// TIA Portal project "Clasificacion de Piezas" (V16)

(* hardware
DEVICE "S71500/ET200MP station_1"  S7-1500 station
   slot 0: "Perfil soporte_0"  Rack  6ES7 590-1***0-0AA0
   slot 1: "PLC_1"  CPU 1512C-1 PN  6ES7 512-1CK00-0AB0  V2.8
      slot 3: "Display de la CPU_1"  6ES7591-1AA00-0AA0
      slot 32768: "Interfaz PROFINET_1"  X1
         slot 32769: "Puerto_1"  X1 P1
         slot 32770: "Puerto_2"  X1 P2
      slot 34817: "Virtual CP interface port_1"  Virtual CP interface port  Virtual CP interface port
DEVICE "HMI_Clasificacion"  KTP900 Basic PN
   slot 0: "HMI_Clasificacion"  KTP900 Basic PN  6AV2 123-2JB03-0AX0  16.0.0.0
   slot 1: "HMI_RT_2"  KTP900 Basic PN  6AV2 123-2JB03-0AX0  16.0.0.0
   slot 5: "HMI_Clasificacion.IE_CP_1"  PROFINET Interface  16.0.0.0
      slot 1: "Interfaz PROFINET_1"  PROFINET Interface
         slot 1: "Port_1"  Port
*)

// ===== PLC "PLC_1"  CPU 1512C-1 PN =====

VAR_GLOBAL   // PLC tag table "Entradas"
   "PM" AT %M0.0 : Bool;   // Pulsador de Macha
   "PP" AT %M0.1 : Bool;   // Pulsador de Paro
   "SE" AT %M0.2 : Bool;   // Seta de Emergencia
   "PR" AT %M0.3 : Bool;   // Pulsador de Rearme
   "FCSuperior" AT %M0.4 : Bool;   // Final de Carrera Superior
   "FCInferior" AT %M0.5 : Bool;   // Final de Carrera Inferior
   "SenCintaEntrada" AT %M0.6 : Bool;   // Sensor de la Cinta de Entrada
   "SenCaja01PosIni" AT %M0.7 : Bool;   // Sensor de la Posición Inicial de la Caja 01
   "SenCaja02PosIni" AT %M1.0 : Bool;   // Sensor de la Posición Inicial de la Caja 02
   "SenCil01Rec" AT %M1.1 : Bool;   // Sensor del Cilindro Recogido
   "SenCil01Med" AT %M1.2 : Bool;   // Sensor del Cilindro en el Medio
   "SenCil01Ext" AT %M1.3 : Bool;   // Sensor del Cilindro Extendido
   "SenIndCaja01" AT %M1.4 : Bool;   // Sensor Inductivo de Giro de la Caja 01
   "SenIndCaja02" AT %M1.5 : Bool;   // Sensor Inductivo de Giro de la Caja 02
   "SenCinta01" AT %M1.6 : Bool;   // Sensor de la Cinta 01
   "SenCinta02" AT %M1.7 : Bool;   // Sensor de la Cinta 02
   "PMAux" AT %M2.0 : Bool;
   "PPAux" AT %M2.1 : Bool;
   "PRAux" AT %M2.2 : Bool;
   "Marcha" AT %M4.4 : Bool;
   "Paro" AT %M4.5 : Bool;
   "Rearme" AT %M4.6 : Bool;
END_VAR

VAR_GLOBAL   // PLC tag table "Salidas"
   "MotorVolteoCaja01Izq" AT %Q0.0 : Bool;   // Motor de Volteo hacia la Izquierda de La Caja 01
   "MotorVolteoCaja01Dch" AT %Q0.1 : Bool;   // Motor de Volteo hacia la Derecha de La Caja 01
   "MotorVolteoCaja02Izq" AT %Q0.2 : Bool;   // Motor de Volteo hacia la Izquierda de La Caja 02
   "MotorVolteoCaja02Dch" AT %Q0.3 : Bool;   // Motor de Volteo hacia la Derecha de La Caja 02
   "MotorCilindroRec" AT %Q0.4 : Bool;   // Motor de Recogida del Cilindro
   "MotorCilindroExt" AT %Q0.5 : Bool;   // Motor de Extension del Cilindro
   "MotorCinta01" AT %Q0.6 : Bool;   // Motor de la Cinta 01
   "MotorCinta02" AT %Q0.7 : Bool;   // Motor de la Cinta 02
   "MotorCintaEntradaAdelante" AT %Q1.0 : Bool;   // Motor de Avance de la Cinta de Entrada
   "MotorCintaEntradaAtras" AT %Q1.1 : Bool;   // Motor de Retroceso de la Cinta de Entrada
   "LV" AT %Q1.2 : Bool;   // Luz Verde
   "LN" AT %Q1.3 : Bool;   // Luz Naranja
   "LR" AT %Q1.4 : Bool;   // Luz Roja
   "LE" AT %Q1.5 : Bool;   // Luz de Emergencia
   "Sirena" AT %Q1.6 : Bool;   // Sirena
END_VAR

VAR_GLOBAL   // PLC tag table "Memorias"
   "Inicio" AT %M2.4 : Bool;
   "SolCondIni" AT %M2.5 : Bool;
   "IniCondIni" AT %M2.6 : Bool;
   "FinCondIni" AT %M2.7 : Bool;
   "ProdNorm" AT %M3.0 : Bool;
   "ParoFC" AT %M3.1 : Bool;
   "InicioCintaEntrada" AT %M3.2 : Bool;
   "InicioRecPiezas" AT %M3.3 : Bool;
   "InicioCinta1" AT %M3.4 : Bool;
   "InicioCinta2" AT %M3.5 : Bool;
   "SolMarchaFin" AT %M3.6 : Bool;
   "IniMarchaFin" AT %M3.7 : Bool;
   "FinMarchaFin" AT %M4.0 : Bool;
   "Emergencia" AT %M4.1 : Bool;
   "PararCintaEntrada" AT %M4.3 : Bool;
   "Timer1" AT %M4.7 : Bool;
   "Cont01" AT %M5.0 : Bool;
   "Cont02" AT %M5.1 : Bool;
   "Timer2" AT %M5.2 : Bool;
   "Timer3" AT %M5.3 : Bool;
   "Timer4" AT %M5.4 : Bool;
END_VAR

DATA_BLOCK "Sec_Principal_DB"   // DB1
{ S7_Optimized_Access := 'TRUE' }
VERSION : 0.1
// stored: InstanceOfName Sec_Principal
"Sec_Principal"
BEGIN
END_DATA_BLOCK

DATA_BLOCK "Recoger_Piezas_DB"   // DB2
{ S7_Optimized_Access := 'TRUE' }
VERSION : 0.1
// stored: InstanceOfName Recoger_Piezas
"Recoger_Piezas"
BEGIN
END_DATA_BLOCK

DATA_BLOCK "Marcha_Fin_DB"   // DB3
{ S7_Optimized_Access := 'TRUE' }
VERSION : 0.1
// stored: InstanceOfName Marcha_Fin
"Marcha_Fin"
BEGIN
END_DATA_BLOCK

DATA_BLOCK "Cond_Ini_DB"   // DB4
{ S7_Optimized_Access := 'TRUE' }
VERSION : 0.1
// stored: InstanceOfName Cond_Ini
"Cond_Ini"
BEGIN
END_DATA_BLOCK

DATA_BLOCK "Cinta_Salida_02_DB"   // DB5
{ S7_Optimized_Access := 'TRUE' }
VERSION : 0.1
// stored: InstanceOfName Cinta_Salida_02
"Cinta_Salida_02"
BEGIN
END_DATA_BLOCK

DATA_BLOCK "Cinta_Salida_01_DB"   // DB6
{ S7_Optimized_Access := 'TRUE' }
VERSION : 0.1
// stored: InstanceOfName Cinta_Salida_01
"Cinta_Salida_01"
BEGIN
END_DATA_BLOCK

DATA_BLOCK "Cinta_Entrada_DB"   // DB7
{ S7_Optimized_Access := 'TRUE' }
VERSION : 0.1
// stored: InstanceOfName Cinta_Entrada
"Cinta_Entrada"
BEGIN
END_DATA_BLOCK

DATA_BLOCK "Paro_Emergencia_DB"   // DB14
{ S7_Optimized_Access := 'TRUE' }
VERSION : 0.1
// stored: InstanceOfName Paro_Emergencia
"Paro_Emergencia"
BEGIN
END_DATA_BLOCK

// folder: System blocks/Program resources

DATA_BLOCK "Timer_1_DB"   // DB8
{ S7_Optimized_Access := 'TRUE' }
AUTHOR : Simatic
FAMILY : IEC
NAME : IEC_TMR
VERSION : 1.0
// stored: InstanceOfName IEC_TIMER
"IEC_TIMER"
BEGIN
END_DATA_BLOCK

DATA_BLOCK "ContCaja01"   // DB9
{ S7_Optimized_Access := 'TRUE' }
AUTHOR : Simatic
FAMILY : IEC
NAME : CNTR
VERSION : 1.0
// stored: InstanceOfName IEC_COUNTER
"IEC_COUNTER"
BEGIN
END_DATA_BLOCK

DATA_BLOCK "ContCaja02"   // DB10
{ S7_Optimized_Access := 'TRUE' }
AUTHOR : Simatic
FAMILY : IEC
NAME : CNTR
VERSION : 1.0
// stored: InstanceOfName IEC_COUNTER
"IEC_COUNTER"
BEGIN
END_DATA_BLOCK

DATA_BLOCK "Timer_2"   // DB11
{ S7_Optimized_Access := 'TRUE' }
AUTHOR : Simatic
FAMILY : IEC
NAME : IEC_TMR
VERSION : 1.0
// stored: InstanceOfName IEC_TIMER
"IEC_TIMER"
BEGIN
END_DATA_BLOCK

DATA_BLOCK "Timer_3"   // DB12
{ S7_Optimized_Access := 'TRUE' }
AUTHOR : Simatic
FAMILY : IEC
NAME : IEC_TMR
VERSION : 1.0
// stored: InstanceOfName IEC_TIMER
"IEC_TIMER"
BEGIN
END_DATA_BLOCK

DATA_BLOCK "Timer_4"   // DB13
{ S7_Optimized_Access := 'TRUE' }
AUTHOR : Simatic
FAMILY : IEC
NAME : IEC_TMR
VERSION : 1.0
// stored: InstanceOfName IEC_TIMER
"IEC_TIMER"
BEGIN
END_DATA_BLOCK

// folder: (top level)

FUNCTION_BLOCK "Sec_Principal"   // FB1, GRAPH_PLUS
{ S7_Optimized_Access := 'TRUE' }
VERSION : 0.1
   VAR_INPUT
      OFF_SQ : Bool := false;   // Desactivar cadena
      INIT_SQ : Bool := false;   // Poner cadena en estado inicial
      ACK_EF : Bool := false;   // Acusar todos los errores y fallos
      S_PREV : Bool := false;   // Mostrar la etapa anterior en el parámetro S_NO
      S_NEXT : Bool := false;   // Mostrar la etapa siguiente en el parámetro S_NO
      SW_AUTO : Bool := false;   // Modo automático
      SW_TAP : Bool := false;   // Semiautomático/continuar con transición
      SW_TOP : Bool := false;   // Semiautomático/transición ignorada
      SW_MAN : Bool := false;   // Modo manual
      S_SEL : Int := 0;   // Seleccionar la etapa que debe mostrarse en S_NO
      S_ON : Bool := false;   // Activar la etapa del parámetro S_NO
      S_OFF : Bool := false;   // Desactivar el incremento presente en el parámetro S_NO
      T_PUSH : Bool := false;   // Habilitar conmutación de transición en modo semiautomático
   END_VAR
   VAR_OUTPUT
      S_NO : Int := 0;   // Número de etapa
      S_MORE : Bool := false;   // Existen más etapas que pueden mostrarse en S_NO.
      S_ACTIVE : Bool := false;   // El incremento presente en el parámetro S_NO está activo
      ERR_FLT : Bool := false;   // Error de grupo interlock o supervisión
      AUTO_ON : Bool := false;   // Modo automático activado
      TAP_ON : Bool := false;   // Modo semiautomático/etapa con transición activada
      TOP_ON : Bool := false;   // Modo semiautomático/Ignorar transición activado
      MAN_ON : Bool := false;   // Modo manual activado
   END_VAR
   VAR
      HMI_INFO : Array[0..8] of UInt;
      IF_PAR : G7_IfParPlus_V6;
      RT_DATA : G7_RTDataPlus_V6;   // Área de datos interna
      Trans1 : G7_TransitionPlus_V6;   // Estructura de la transición
      Trans2 : G7_TransitionPlus_V6;   // Estructura de la transición
      Trans3 : G7_TransitionPlus_V6;   // Estructura de la transición
      Trans4 : G7_TransitionPlus_V6;   // Estructura de la transición
      Trans5 : G7_TransitionPlus_V6;   // Estructura de la transición
      X0 : G7_StepPlus_V6;   // Estructura de la etapa
      X1 : G7_StepPlus_V6;   // Estructura de la etapa
      X2 : G7_StepPlus_V6;   // Estructura de la etapa
      X3 : G7_StepPlus_V6;   // Estructura de la etapa
      X4 : G7_StepPlus_V6;   // Estructura de la etapa
      SINI : Array[0..1] of USInt;
      LSTT : Array[0..4] of USInt;
      ATAJ : Array[0..4] of USInt;
      ATAB : Array[0..4] of USInt;
      PSTT : Array[0..4] of USInt;
      NSTT : Array[0..4] of USInt;
      ASSJ : Array[0..4] of USInt;
      ASSB : Array[0..4] of USInt;
      PTTS : Array[0..4] of USInt;
      NTTS : Array[0..4] of USInt;
      SW_SQTS : Array[0..4] of USInt;
      SWITCH : Array[0..0] of USInt;
      TVX : Array[0..1] of USInt;
      TTX : Array[0..1] of USInt;
      TSX : Array[0..1] of USInt;
      S00X : Array[0..1] of USInt;
      SOFFX : Array[0..1] of USInt;
      SONX : Array[0..1] of USInt;
      SAX : Array[0..1] of USInt;
      SERRX : Array[0..5] of USInt;
      SMX : Array[0..5] of USInt;
      S0X : Array[0..5] of USInt;
      S1X : Array[0..5] of USInt;
      IL_ALARM_INST : Diag_Alarm;
      SUP_ALARM_INST : Diag_Alarm;
      STEP_TIME_ALARM_INST : Diag_Alarm;
      IEC_TIMER_INST : IEC_TIMER;
      TRANSACTION_FLAG : Bool := false;
   END_VAR
   // SINI[0] := 2;
   // LSTT[0] := 255;
   // LSTT[1] := 255;
   // LSTT[2] := 255;
   // LSTT[3] := 255;
   // ATAJ[1] := 1;
   // ATAJ[2] := 2;
   // ATAJ[3] := 3;
   // ATAJ[4] := 4;
   // ATAB[1] := 1;
   // ATAB[2] := 2;
   // ATAB[3] := 3;
   // ATAB[4] := 4;
   // PSTT[0] := 1;
   // PSTT[2] := 2;
   // PSTT[3] := 3;
   // PSTT[4] := 4;
   // NSTT[0] := 2;
   // NSTT[1] := 1;
   // NSTT[2] := 3;
   // NSTT[3] := 4;
   // ASSJ[1] := 1;
   // ASSJ[2] := 2;
   // ASSJ[3] := 3;
   // ASSJ[4] := 4;
   // ASSB[1] := 1;
   // ASSB[2] := 2;
   // ASSB[3] := 3;
   // ASSB[4] := 4;
   // PTTS[0] := 255;
   // PTTS[1] := 1;
   // PTTS[3] := 2;
   // PTTS[4] := 3;
   // NTTS[0] := 1;
   // NTTS[2] := 2;
   // NTTS[3] := 3;
   // NTTS[4] := 4;
   // TVX[0] := 16#1;
   // TTX[0] := 16#1;
   // TSX[0] := 16#1;
   // S00X[0] := 16#1;
   // SOFFX[0] := 16#1;
   // SONX[0] := 16#1;
   // SAX[0] := 16#1;
   // SERRX[0] := 16#1;
   // SMX[0] := 16#1;
   // S0X[0] := 16#1;
   // S1X[0] := 16#1;
BEGIN
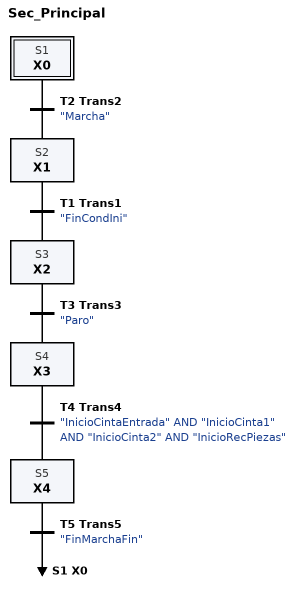
   // sequencer 1
   INITIAL_STEP X0:   // S1, max time T#10S, warning time T#7S
   END_STEP
   TRANSITION Trans2 FROM X0 TO X1   // T2
      := "Marcha";
   END_TRANSITION
   STEP X1:   // S2, max time T#10S, warning time T#7S
   END_STEP
   TRANSITION Trans1 FROM X1 TO X2   // T1
      := "FinCondIni";
   END_TRANSITION
   STEP X2:   // S3, max time T#10S, warning time T#7S
   END_STEP
   TRANSITION Trans3 FROM X2 TO X3   // T3
      := "Paro";
   END_TRANSITION
   STEP X3:   // S4, max time T#10S, warning time T#7S
   END_STEP
   TRANSITION Trans4 FROM X3 TO X4   // T4
      := "InicioCintaEntrada" AND "InicioCinta1" AND "InicioCinta2" AND "InicioRecPiezas";
   END_TRANSITION
   STEP X4:   // S5, max time T#10S, warning time T#7S
   END_STEP
   TRANSITION Trans5 FROM X4 TO X0   // T5, jump
      := "FinMarchaFin";
   END_TRANSITION
END_FUNCTION_BLOCK

FUNCTION_BLOCK "Cond_Ini"   // FB2, GRAPH_PLUS
{ S7_Optimized_Access := 'TRUE' }
VERSION : 0.1
   VAR_INPUT
      OFF_SQ : Bool := false;   // Desactivar cadena
      INIT_SQ : Bool := false;   // Poner cadena en estado inicial
      ACK_EF : Bool := false;   // Acusar todos los errores y fallos
      S_PREV : Bool := false;   // Mostrar la etapa anterior en el parámetro S_NO
      S_NEXT : Bool := false;   // Mostrar la etapa siguiente en el parámetro S_NO
      SW_AUTO : Bool := false;   // Modo automático
      SW_TAP : Bool := false;   // Semiautomático/continuar con transición
      SW_TOP : Bool := false;   // Semiautomático/transición ignorada
      SW_MAN : Bool := false;   // Modo manual
      S_SEL : Int := 0;   // Seleccionar la etapa que debe mostrarse en S_NO
      S_ON : Bool := false;   // Activar la etapa del parámetro S_NO
      S_OFF : Bool := false;   // Desactivar el incremento presente en el parámetro S_NO
      T_PUSH : Bool := false;   // Habilitar conmutación de transición en modo semiautomático
   END_VAR
   VAR_OUTPUT
      S_NO : Int := 0;   // Número de etapa
      S_MORE : Bool := false;   // Existen más etapas que pueden mostrarse en S_NO.
      S_ACTIVE : Bool := false;   // El incremento presente en el parámetro S_NO está activo
      ERR_FLT : Bool := false;   // Error de grupo interlock o supervisión
      AUTO_ON : Bool := false;   // Modo automático activado
      TAP_ON : Bool := false;   // Modo semiautomático/etapa con transición activada
      TOP_ON : Bool := false;   // Modo semiautomático/Ignorar transición activado
      MAN_ON : Bool := false;   // Modo manual activado
   END_VAR
   VAR
      HMI_INFO : Array[0..13] of UInt;
      IF_PAR : G7_IfParPlus_V6;
      RT_DATA : G7_RTDataPlus_V6;   // Área de datos interna
      Trans1 : G7_TransitionPlus_V6;   // Estructura de la transición
      Trans2 : G7_TransitionPlus_V6;   // Estructura de la transición
      Trans3 : G7_TransitionPlus_V6;   // Estructura de la transición
      Trans4 : G7_TransitionPlus_V6;   // Estructura de la transición
      Trans5 : G7_TransitionPlus_V6;   // Estructura de la transición
      Trans6 : G7_TransitionPlus_V6;   // Estructura de la transición
      Trans7 : G7_TransitionPlus_V6;   // Estructura de la transición
      Trans8 : G7_TransitionPlus_V6;   // Estructura de la transición
      Trans9 : G7_TransitionPlus_V6;   // Estructura de la transición
      Trans10 : G7_TransitionPlus_V6;   // Estructura de la transición
      Trans11 : G7_TransitionPlus_V6;   // Estructura de la transición
      X10 : G7_StepPlus_V6;   // Estructura de la etapa
      X13 : G7_StepPlus_V6;   // Estructura de la etapa
      X14 : G7_StepPlus_V6;   // Estructura de la etapa
      X15 : G7_StepPlus_V6;   // Estructura de la etapa
      X16 : G7_StepPlus_V6;   // Estructura de la etapa
      X11 : G7_StepPlus_V6;   // Estructura de la etapa
      X12 : G7_StepPlus_V6;   // Estructura de la etapa
      X19 : G7_StepPlus_V6;   // Estructura de la etapa
      X21 : G7_StepPlus_V6;   // Estructura de la etapa
      X17 : G7_StepPlus_V6;   // Estructura de la etapa
      X18 : G7_StepPlus_V6;   // Estructura de la etapa
      X20 : G7_StepPlus_V6;   // Estructura de la etapa
      X22 : G7_StepPlus_V6;   // Estructura de la etapa
      X23 : G7_StepPlus_V6;   // Estructura de la etapa
      SINI : Array[0..6] of USInt;
      LSTT : Array[0..10] of USInt;
      ATAJ : Array[0..10] of USInt;
      ATAB : Array[0..10] of USInt;
      PSTT : Array[0..10] of USInt;
      NSTT : Array[0..10] of USInt;
      ASSJ : Array[0..13] of USInt;
      ASSB : Array[0..13] of USInt;
      PTTS : Array[0..13] of USInt;
      NTTS : Array[0..13] of USInt;
      SW_SQTS : Array[0..13] of USInt;
      SWITCH : Array[0..6] of USInt;
      TVX : Array[0..6] of USInt;
      TTX : Array[0..6] of USInt;
      TSX : Array[0..6] of USInt;
      S00X : Array[0..6] of USInt;
      SOFFX : Array[0..6] of USInt;
      SONX : Array[0..6] of USInt;
      SAX : Array[0..6] of USInt;
      SERRX : Array[0..14] of USInt;
      SMX : Array[0..14] of USInt;
      S0X : Array[0..14] of USInt;
      S1X : Array[0..14] of USInt;
      IL_ALARM_INST : Diag_Alarm;
      SUP_ALARM_INST : Diag_Alarm;
      STEP_TIME_ALARM_INST : Diag_Alarm;
      IEC_TIMER_INST : IEC_TIMER;
      TRANSACTION_FLAG : Bool := false;
   END_VAR
   // SINI[0] := 2;
   // SINI[2] := 255;
   // SINI[3] := 255;
   // SINI[4] := 255;
   // SINI[5] := 255;
   // SINI[6] := 255;
   // LSTT[0] := 255;
   // LSTT[1] := 255;
   // LSTT[2] := 255;
   // LSTT[3] := 255;
   // LSTT[4] := 255;
   // LSTT[5] := 255;
   // LSTT[6] := 255;
   // LSTT[7] := 255;
   // LSTT[8] := 255;
   // LSTT[9] := 255;
   // ATAJ[1] := 1;
   // ATAJ[2] := 2;
   // ATAJ[3] := 3;
   // ATAJ[4] := 4;
   // ATAJ[5] := 5;
   // ATAJ[6] := 6;
   // ATAJ[7] := 7;
   // ATAJ[8] := 8;
   // ATAJ[9] := 9;
   // ATAJ[10] := 10;
   // ATAB[1] := 1;
   // ATAB[2] := 2;
   // ATAB[3] := 3;
   // ATAB[4] := 4;
   // ATAB[5] := 5;
   // ATAB[6] := 6;
   // ATAB[7] := 7;
   // ATAB[8] := 8;
   // ATAB[9] := 9;
   // ATAB[10] := 10;
   // PSTT[1] := 1;
   // PSTT[2] := 2;
   // PSTT[3] := 3;
   // PSTT[4] := 5;
   // PSTT[5] := 4;
   // PSTT[6] := 9;
   // PSTT[7] := 7;
   // PSTT[8] := 8;
   // PSTT[9] := 6;
   // PSTT[10] := 13;
   // NSTT[0] := 5;
   // NSTT[1] := 2;
   // NSTT[2] := 3;
   // NSTT[3] := 4;
   // NSTT[4] := 6;
   // NSTT[5] := 9;
   // NSTT[6] := 10;
   // NSTT[7] := 11;
   // NSTT[8] := 12;
   // NSTT[9] := 13;
   // ASSJ[1] := 1;
   // ASSJ[2] := 2;
   // ASSJ[3] := 3;
   // ASSJ[4] := 4;
   // ASSJ[5] := 5;
   // ASSJ[6] := 10;
   // ASSJ[7] := 7;
   // ASSJ[8] := 8;
   // ASSJ[9] := 9;
   // ASSJ[10] := 11;
   // ASSJ[11] := 12;
   // ASSJ[12] := 6;
   // ASSJ[13] := 13;
   // ASSB[1] := 5;
   // ASSB[2] := 2;
   // ASSB[3] := 3;
   // ASSB[4] := 4;
   // ASSB[5] := 1;
   // ASSB[6] := 6;
   // ASSB[7] := 8;
   // ASSB[8] := 9;
   // ASSB[9] := 7;
   // ASSB[10] := 10;
   // ASSB[11] := 11;
   // ASSB[12] := 12;
   // ASSB[13] := 13;
   // PTTS[0] := 255;
   // PTTS[2] := 1;
   // PTTS[3] := 2;
   // PTTS[4] := 3;
   // PTTS[6] := 4;
   // PTTS[7] := 5;
   // PTTS[8] := 5;
   // PTTS[9] := 5;
   // PTTS[10] := 6;
   // PTTS[11] := 7;
   // PTTS[12] := 8;
   // PTTS[13] := 9;
   // NTTS[1] := 1;
   // NTTS[2] := 2;
   // NTTS[3] := 3;
   // NTTS[4] := 5;
   // NTTS[5] := 4;
   // NTTS[6] := 9;
   // NTTS[7] := 7;
   // NTTS[8] := 8;
   // NTTS[9] := 6;
   // NTTS[10] := 9;
   // NTTS[11] := 9;
   // NTTS[12] := 9;
   // NTTS[13] := 10;
   // SW_SQTS[1] := 1;
   // SW_SQTS[2] := 1;
   // SW_SQTS[3] := 1;
   // SW_SQTS[4] := 1;
   // SW_SQTS[5] := 2;
   // SW_SQTS[6] := 2;
   // SW_SQTS[7] := 3;
   // SW_SQTS[8] := 4;
   // SW_SQTS[9] := 5;
   // SW_SQTS[10] := 5;
   // SW_SQTS[11] := 3;
   // SW_SQTS[12] := 4;
   // SW_SQTS[13] := 6;
   // SWITCH[1] := 130;
   // SWITCH[2] := 142;
   // SWITCH[3] := 198;
   // SWITCH[4] := 226;
   // TVX[0] := 16#1;
   // TTX[0] := 16#1;
   // TSX[0] := 16#1;
   // S00X[0] := 16#1;
   // SOFFX[0] := 16#1;
   // SONX[0] := 16#1;
   // SAX[0] := 16#1;
   // SERRX[0] := 16#1;
   // SMX[0] := 16#1;
   // S0X[0] := 16#1;
   // S1X[0] := 16#1;
BEGIN
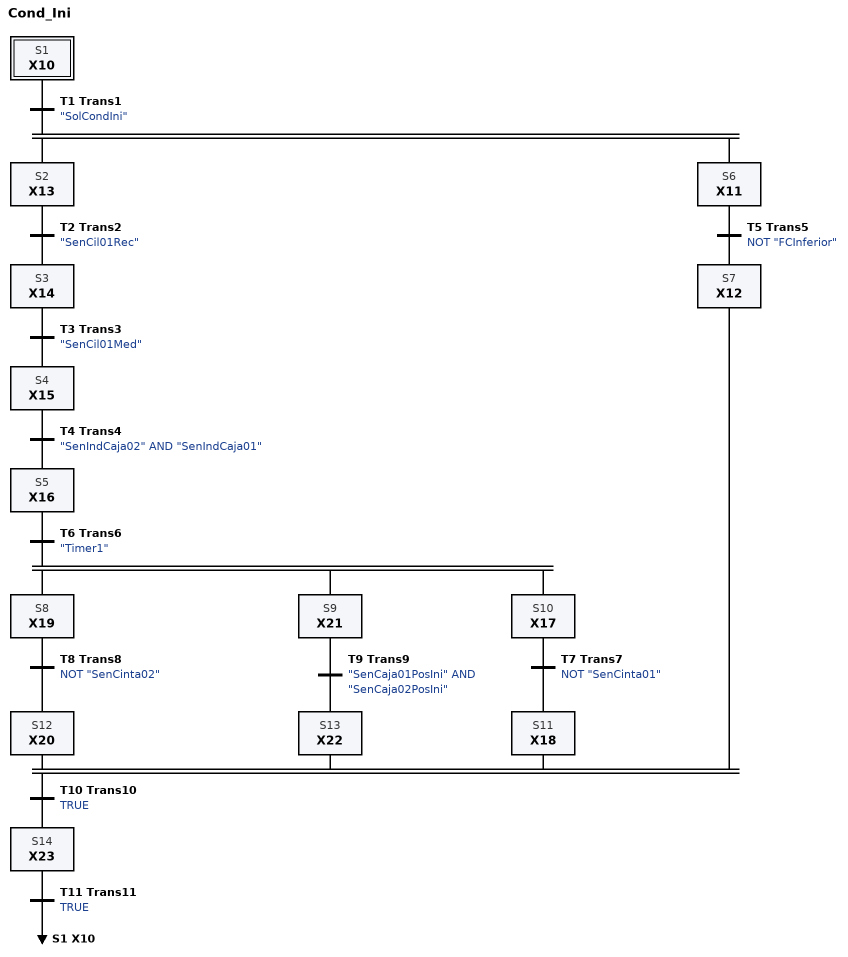
   // sequencer 1
   INITIAL_STEP X10:   // S1, max time T#10S, warning time T#7S
   END_STEP
   TRANSITION Trans1 FROM X10 TO (X13, X11)   // T1
      := "SolCondIni";
   END_TRANSITION
   STEP X13:   // S2, max time T#10S, warning time T#7S
   END_STEP
   TRANSITION Trans2 FROM X13 TO X14   // T2
      := "SenCil01Rec";
   END_TRANSITION
   STEP X14:   // S3, max time T#10S, warning time T#7S
   END_STEP
   TRANSITION Trans3 FROM X14 TO X15   // T3
      := "SenCil01Med";
   END_TRANSITION
   STEP X15:   // S4, max time T#10S, warning time T#7S
   END_STEP
   TRANSITION Trans4 FROM X15 TO X16   // T4
      := "SenIndCaja02" AND "SenIndCaja01";
   END_TRANSITION
   STEP X16:   // S5, max time T#10S, warning time T#7S
   END_STEP
   TRANSITION Trans6 FROM X16 TO (X19, X21, X17)   // T6
      := "Timer1";
   END_TRANSITION
   STEP X11:   // S6, max time T#10S, warning time T#7S
   END_STEP
   TRANSITION Trans5 FROM X11 TO X12   // T5
      := NOT "FCInferior";
   END_TRANSITION
   STEP X12:   // S7, max time T#10S, warning time T#7S
   END_STEP
   STEP X19:   // S8, max time T#10S, warning time T#7S
   END_STEP
   TRANSITION Trans8 FROM X19 TO X20   // T8
      := NOT "SenCinta02";
   END_TRANSITION
   STEP X21:   // S9, max time T#10S, warning time T#7S
   END_STEP
   TRANSITION Trans9 FROM X21 TO X22   // T9
      := "SenCaja01PosIni" AND "SenCaja02PosIni";
   END_TRANSITION
   STEP X17:   // S10, max time T#10S, warning time T#7S
   END_STEP
   TRANSITION Trans7 FROM X17 TO X18   // T7
      := NOT "SenCinta01";
   END_TRANSITION
   STEP X18:   // S11, max time T#10S, warning time T#7S
   END_STEP
   STEP X20:   // S12, max time T#10S, warning time T#7S
   END_STEP
   TRANSITION Trans10 FROM (X12, X22, X18, X20) TO X23   // T10
      := TRUE;
   END_TRANSITION
   STEP X22:   // S13, max time T#10S, warning time T#7S
   END_STEP
   STEP X23:   // S14, max time T#10S, warning time T#7S
   END_STEP
   TRANSITION Trans11 FROM X23 TO X10   // T11, jump
      := TRUE;
   END_TRANSITION
END_FUNCTION_BLOCK

FUNCTION_BLOCK "Cinta_Entrada"   // FB3, GRAPH_PLUS
{ S7_Optimized_Access := 'TRUE' }
VERSION : 0.1
   VAR_INPUT
      OFF_SQ : Bool := false;   // Desactivar cadena
      INIT_SQ : Bool := false;   // Poner cadena en estado inicial
      ACK_EF : Bool := false;   // Acusar todos los errores y fallos
      S_PREV : Bool := false;   // Mostrar la etapa anterior en el parámetro S_NO
      S_NEXT : Bool := false;   // Mostrar la etapa siguiente en el parámetro S_NO
      SW_AUTO : Bool := false;   // Modo automático
      SW_TAP : Bool := false;   // Semiautomático/continuar con transición
      SW_TOP : Bool := false;   // Semiautomático/transición ignorada
      SW_MAN : Bool := false;   // Modo manual
      S_SEL : Int := 0;   // Seleccionar la etapa que debe mostrarse en S_NO
      S_ON : Bool := false;   // Activar la etapa del parámetro S_NO
      S_OFF : Bool := false;   // Desactivar el incremento presente en el parámetro S_NO
      T_PUSH : Bool := false;   // Habilitar conmutación de transición en modo semiautomático
   END_VAR
   VAR_OUTPUT
      S_NO : Int := 0;   // Número de etapa
      S_MORE : Bool := false;   // Existen más etapas que pueden mostrarse en S_NO.
      S_ACTIVE : Bool := false;   // El incremento presente en el parámetro S_NO está activo
      ERR_FLT : Bool := false;   // Error de grupo interlock o supervisión
      AUTO_ON : Bool := false;   // Modo automático activado
      TAP_ON : Bool := false;   // Modo semiautomático/etapa con transición activada
      TOP_ON : Bool := false;   // Modo semiautomático/Ignorar transición activado
      MAN_ON : Bool := false;   // Modo manual activado
   END_VAR
   VAR
      HMI_INFO : Array[0..8] of UInt;
      IF_PAR : G7_IfParPlus_V6;
      RT_DATA : G7_RTDataPlus_V6;   // Área de datos interna
      Trans1 : G7_TransitionPlus_V6;   // Estructura de la transición
      Trans2 : G7_TransitionPlus_V6;   // Estructura de la transición
      X30 : G7_StepPlus_V6;   // Estructura de la etapa
      X31 : G7_StepPlus_V6;   // Estructura de la etapa
      SINI : Array[0..1] of USInt;
      LSTT : Array[0..1] of USInt;
      ATAJ : Array[0..1] of USInt;
      ATAB : Array[0..1] of USInt;
      PSTT : Array[0..1] of USInt;
      NSTT : Array[0..1] of USInt;
      ASSJ : Array[0..1] of USInt;
      ASSB : Array[0..1] of USInt;
      PTTS : Array[0..1] of USInt;
      NTTS : Array[0..1] of USInt;
      SW_SQTS : Array[0..1] of USInt;
      SWITCH : Array[0..0] of USInt;
      TVX : Array[0..1] of USInt;
      TTX : Array[0..1] of USInt;
      TSX : Array[0..1] of USInt;
      S00X : Array[0..1] of USInt;
      SOFFX : Array[0..1] of USInt;
      SONX : Array[0..1] of USInt;
      SAX : Array[0..1] of USInt;
      SERRX : Array[0..2] of USInt;
      SMX : Array[0..2] of USInt;
      S0X : Array[0..2] of USInt;
      S1X : Array[0..2] of USInt;
      IL_ALARM_INST : Diag_Alarm;
      SUP_ALARM_INST : Diag_Alarm;
      STEP_TIME_ALARM_INST : Diag_Alarm;
      IEC_TIMER_INST : IEC_TIMER;
      TRANSACTION_FLAG : Bool := false;
   END_VAR
   // SINI[0] := 2;
   // LSTT[0] := 255;
   // ATAJ[1] := 1;
   // ATAB[1] := 1;
   // PSTT[1] := 1;
   // NSTT[0] := 1;
   // ASSJ[1] := 1;
   // ASSB[1] := 1;
   // PTTS[0] := 255;
   // NTTS[1] := 1;
   // TVX[0] := 16#1;
   // TTX[0] := 16#1;
   // TSX[0] := 16#1;
   // S00X[0] := 16#1;
   // SOFFX[0] := 16#1;
   // SONX[0] := 16#1;
   // SAX[0] := 16#1;
   // SERRX[0] := 16#1;
   // SMX[0] := 16#1;
   // S0X[0] := 16#1;
   // S1X[0] := 16#1;
BEGIN
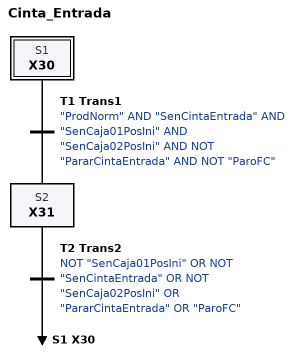
   // sequencer 1
   INITIAL_STEP X30:   // S1, max time T#10S, warning time T#7S
   END_STEP
   TRANSITION Trans1 FROM X30 TO X31   // T1
      := "ProdNorm" AND "SenCintaEntrada" AND "SenCaja01PosIni" AND "SenCaja02PosIni" AND NOT "PararCintaEntrada" AND NOT "ParoFC";
   END_TRANSITION
   STEP X31:   // S2, max time T#10S, warning time T#7S
   END_STEP
   TRANSITION Trans2 FROM X31 TO X30   // T2, jump
      := NOT "SenCaja01PosIni" OR NOT "SenCintaEntrada" OR NOT "SenCaja02PosIni" OR "PararCintaEntrada" OR "ParoFC";
   END_TRANSITION
END_FUNCTION_BLOCK

FUNCTION_BLOCK "Cinta_Salida_01"   // FB4, GRAPH_PLUS
{ S7_Optimized_Access := 'TRUE' }
VERSION : 0.1
   VAR_INPUT
      OFF_SQ : Bool := false;   // Desactivar cadena
      INIT_SQ : Bool := false;   // Poner cadena en estado inicial
      ACK_EF : Bool := false;   // Acusar todos los errores y fallos
      S_PREV : Bool := false;   // Mostrar la etapa anterior en el parámetro S_NO
      S_NEXT : Bool := false;   // Mostrar la etapa siguiente en el parámetro S_NO
      SW_AUTO : Bool := false;   // Modo automático
      SW_TAP : Bool := false;   // Semiautomático/continuar con transición
      SW_TOP : Bool := false;   // Semiautomático/transición ignorada
      SW_MAN : Bool := false;   // Modo manual
      S_SEL : Int := 0;   // Seleccionar la etapa que debe mostrarse en S_NO
      S_ON : Bool := false;   // Activar la etapa del parámetro S_NO
      S_OFF : Bool := false;   // Desactivar el incremento presente en el parámetro S_NO
      T_PUSH : Bool := false;   // Habilitar conmutación de transición en modo semiautomático
   END_VAR
   VAR_OUTPUT
      S_NO : Int := 0;   // Número de etapa
      S_MORE : Bool := false;   // Existen más etapas que pueden mostrarse en S_NO.
      S_ACTIVE : Bool := false;   // El incremento presente en el parámetro S_NO está activo
      ERR_FLT : Bool := false;   // Error de grupo interlock o supervisión
      AUTO_ON : Bool := false;   // Modo automático activado
      TAP_ON : Bool := false;   // Modo semiautomático/etapa con transición activada
      TOP_ON : Bool := false;   // Modo semiautomático/Ignorar transición activado
      MAN_ON : Bool := false;   // Modo manual activado
   END_VAR
   VAR
      HMI_INFO : Array[0..8] of UInt;
      IF_PAR : G7_IfParPlus_V6;
      RT_DATA : G7_RTDataPlus_V6;   // Área de datos interna
      Trans1 : G7_TransitionPlus_V6;   // Estructura de la transición
      Trans2 : G7_TransitionPlus_V6;   // Estructura de la transición
      X60 : G7_StepPlus_V6;   // Estructura de la etapa
      X61 : G7_StepPlus_V6;   // Estructura de la etapa
      SINI : Array[0..1] of USInt;
      LSTT : Array[0..1] of USInt;
      ATAJ : Array[0..1] of USInt;
      ATAB : Array[0..1] of USInt;
      PSTT : Array[0..1] of USInt;
      NSTT : Array[0..1] of USInt;
      ASSJ : Array[0..1] of USInt;
      ASSB : Array[0..1] of USInt;
      PTTS : Array[0..1] of USInt;
      NTTS : Array[0..1] of USInt;
      SW_SQTS : Array[0..1] of USInt;
      SWITCH : Array[0..0] of USInt;
      TVX : Array[0..1] of USInt;
      TTX : Array[0..1] of USInt;
      TSX : Array[0..1] of USInt;
      S00X : Array[0..1] of USInt;
      SOFFX : Array[0..1] of USInt;
      SONX : Array[0..1] of USInt;
      SAX : Array[0..1] of USInt;
      SERRX : Array[0..2] of USInt;
      SMX : Array[0..2] of USInt;
      S0X : Array[0..2] of USInt;
      S1X : Array[0..2] of USInt;
      IL_ALARM_INST : Diag_Alarm;
      SUP_ALARM_INST : Diag_Alarm;
      STEP_TIME_ALARM_INST : Diag_Alarm;
      IEC_TIMER_INST : IEC_TIMER;
      TRANSACTION_FLAG : Bool := false;
   END_VAR
   // SINI[0] := 2;
   // LSTT[0] := 255;
   // ATAJ[1] := 1;
   // ATAB[1] := 1;
   // PSTT[1] := 1;
   // NSTT[0] := 1;
   // ASSJ[1] := 1;
   // ASSB[1] := 1;
   // PTTS[0] := 255;
   // NTTS[1] := 1;
   // TVX[0] := 16#1;
   // TTX[0] := 16#1;
   // TSX[0] := 16#1;
   // S00X[0] := 16#1;
   // SOFFX[0] := 16#1;
   // SONX[0] := 16#1;
   // SAX[0] := 16#1;
   // SERRX[0] := 16#1;
   // SMX[0] := 16#1;
   // S0X[0] := 16#1;
   // S1X[0] := 16#1;
BEGIN
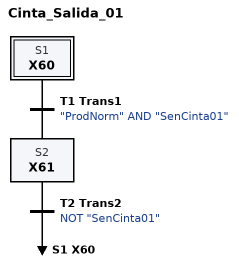
   // sequencer 1
   INITIAL_STEP X60:   // S1, max time T#10S, warning time T#7S
   END_STEP
   TRANSITION Trans1 FROM X60 TO X61   // T1
      := "ProdNorm" AND "SenCinta01";
   END_TRANSITION
   STEP X61:   // S2, max time T#10S, warning time T#7S
   END_STEP
   TRANSITION Trans2 FROM X61 TO X60   // T2, jump
      := NOT "SenCinta01";
   END_TRANSITION
END_FUNCTION_BLOCK

FUNCTION_BLOCK "Cinta_Salida_02"   // FB5, GRAPH_PLUS
{ S7_Optimized_Access := 'TRUE' }
VERSION : 0.1
   VAR_INPUT
      OFF_SQ : Bool := false;   // Desactivar cadena
      INIT_SQ : Bool := false;   // Poner cadena en estado inicial
      ACK_EF : Bool := false;   // Acusar todos los errores y fallos
      S_PREV : Bool := false;   // Mostrar la etapa anterior en el parámetro S_NO
      S_NEXT : Bool := false;   // Mostrar la etapa siguiente en el parámetro S_NO
      SW_AUTO : Bool := false;   // Modo automático
      SW_TAP : Bool := false;   // Semiautomático/continuar con transición
      SW_TOP : Bool := false;   // Semiautomático/transición ignorada
      SW_MAN : Bool := false;   // Modo manual
      S_SEL : Int := 0;   // Seleccionar la etapa que debe mostrarse en S_NO
      S_ON : Bool := false;   // Activar la etapa del parámetro S_NO
      S_OFF : Bool := false;   // Desactivar el incremento presente en el parámetro S_NO
      T_PUSH : Bool := false;   // Habilitar conmutación de transición en modo semiautomático
   END_VAR
   VAR_OUTPUT
      S_NO : Int := 0;   // Número de etapa
      S_MORE : Bool := false;   // Existen más etapas que pueden mostrarse en S_NO.
      S_ACTIVE : Bool := false;   // El incremento presente en el parámetro S_NO está activo
      ERR_FLT : Bool := false;   // Error de grupo interlock o supervisión
      AUTO_ON : Bool := false;   // Modo automático activado
      TAP_ON : Bool := false;   // Modo semiautomático/etapa con transición activada
      TOP_ON : Bool := false;   // Modo semiautomático/Ignorar transición activado
      MAN_ON : Bool := false;   // Modo manual activado
   END_VAR
   VAR
      HMI_INFO : Array[0..8] of UInt;
      IF_PAR : G7_IfParPlus_V6;
      RT_DATA : G7_RTDataPlus_V6;   // Área de datos interna
      Trans1 : G7_TransitionPlus_V6;   // Estructura de la transición
      Trans2 : G7_TransitionPlus_V6;   // Estructura de la transición
      X70 : G7_StepPlus_V6;   // Estructura de la etapa
      X71 : G7_StepPlus_V6;   // Estructura de la etapa
      SINI : Array[0..1] of USInt;
      LSTT : Array[0..1] of USInt;
      ATAJ : Array[0..1] of USInt;
      ATAB : Array[0..1] of USInt;
      PSTT : Array[0..1] of USInt;
      NSTT : Array[0..1] of USInt;
      ASSJ : Array[0..1] of USInt;
      ASSB : Array[0..1] of USInt;
      PTTS : Array[0..1] of USInt;
      NTTS : Array[0..1] of USInt;
      SW_SQTS : Array[0..1] of USInt;
      SWITCH : Array[0..0] of USInt;
      TVX : Array[0..1] of USInt;
      TTX : Array[0..1] of USInt;
      TSX : Array[0..1] of USInt;
      S00X : Array[0..1] of USInt;
      SOFFX : Array[0..1] of USInt;
      SONX : Array[0..1] of USInt;
      SAX : Array[0..1] of USInt;
      SERRX : Array[0..2] of USInt;
      SMX : Array[0..2] of USInt;
      S0X : Array[0..2] of USInt;
      S1X : Array[0..2] of USInt;
      IL_ALARM_INST : Diag_Alarm;
      SUP_ALARM_INST : Diag_Alarm;
      STEP_TIME_ALARM_INST : Diag_Alarm;
      IEC_TIMER_INST : IEC_TIMER;
      TRANSACTION_FLAG : Bool := false;
   END_VAR
   // SINI[0] := 2;
   // LSTT[0] := 255;
   // ATAJ[1] := 1;
   // ATAB[1] := 1;
   // PSTT[1] := 1;
   // NSTT[0] := 1;
   // ASSJ[1] := 1;
   // ASSB[1] := 1;
   // PTTS[0] := 255;
   // NTTS[1] := 1;
   // TVX[0] := 16#1;
   // TTX[0] := 16#1;
   // TSX[0] := 16#1;
   // S00X[0] := 16#1;
   // SOFFX[0] := 16#1;
   // SONX[0] := 16#1;
   // SAX[0] := 16#1;
   // SERRX[0] := 16#1;
   // SMX[0] := 16#1;
   // S0X[0] := 16#1;
   // S1X[0] := 16#1;
BEGIN
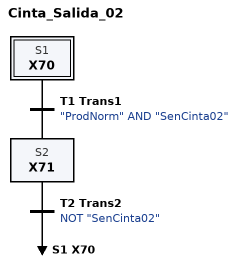
   // sequencer 1
   INITIAL_STEP X70:   // S1, max time T#10S, warning time T#7S
   END_STEP
   TRANSITION Trans1 FROM X70 TO X71   // T1
      := "ProdNorm" AND "SenCinta02";
   END_TRANSITION
   STEP X71:   // S2, max time T#10S, warning time T#7S
   END_STEP
   TRANSITION Trans2 FROM X71 TO X70   // T2, jump
      := NOT "SenCinta02";
   END_TRANSITION
END_FUNCTION_BLOCK

FUNCTION_BLOCK "Recoger_Piezas"   // FB6, GRAPH_PLUS
{ S7_Optimized_Access := 'TRUE' }
VERSION : 0.1
   VAR_INPUT
      OFF_SQ : Bool := false;   // Desactivar cadena
      INIT_SQ : Bool := false;   // Poner cadena en estado inicial
      ACK_EF : Bool := false;   // Acusar todos los errores y fallos
      S_PREV : Bool := false;   // Mostrar la etapa anterior en el parámetro S_NO
      S_NEXT : Bool := false;   // Mostrar la etapa siguiente en el parámetro S_NO
      SW_AUTO : Bool := false;   // Modo automático
      SW_TAP : Bool := false;   // Semiautomático/continuar con transición
      SW_TOP : Bool := false;   // Semiautomático/transición ignorada
      SW_MAN : Bool := false;   // Modo manual
      S_SEL : Int := 0;   // Seleccionar la etapa que debe mostrarse en S_NO
      S_ON : Bool := false;   // Activar la etapa del parámetro S_NO
      S_OFF : Bool := false;   // Desactivar el incremento presente en el parámetro S_NO
      T_PUSH : Bool := false;   // Habilitar conmutación de transición en modo semiautomático
   END_VAR
   VAR_OUTPUT
      S_NO : Int := 0;   // Número de etapa
      S_MORE : Bool := false;   // Existen más etapas que pueden mostrarse en S_NO.
      S_ACTIVE : Bool := false;   // El incremento presente en el parámetro S_NO está activo
      ERR_FLT : Bool := false;   // Error de grupo interlock o supervisión
      AUTO_ON : Bool := false;   // Modo automático activado
      TAP_ON : Bool := false;   // Modo semiautomático/etapa con transición activada
      TOP_ON : Bool := false;   // Modo semiautomático/Ignorar transición activado
      MAN_ON : Bool := false;   // Modo manual activado
   END_VAR
   VAR
      HMI_INFO : Array[0..8] of UInt;
      IF_PAR : G7_IfParPlus_V6;
      RT_DATA : G7_RTDataPlus_V6;   // Área de datos interna
      Trans1 : G7_TransitionPlus_V6;   // Estructura de la transición
      Trans2 : G7_TransitionPlus_V6;   // Estructura de la transición
      Trans3 : G7_TransitionPlus_V6;   // Estructura de la transición
      Trans4 : G7_TransitionPlus_V6;   // Estructura de la transición
      Trans5 : G7_TransitionPlus_V6;   // Estructura de la transición
      Trans6 : G7_TransitionPlus_V6;   // Estructura de la transición
      Trans7 : G7_TransitionPlus_V6;   // Estructura de la transición
      Trans8 : G7_TransitionPlus_V6;   // Estructura de la transición
      Trans9 : G7_TransitionPlus_V6;   // Estructura de la transición
      Trans10 : G7_TransitionPlus_V6;   // Estructura de la transición
      Trans11 : G7_TransitionPlus_V6;   // Estructura de la transición
      Trans13 : G7_TransitionPlus_V6;   // Estructura de la transición
      Trans14 : G7_TransitionPlus_V6;   // Estructura de la transición
      Trans15 : G7_TransitionPlus_V6;   // Estructura de la transición
      Trans16 : G7_TransitionPlus_V6;   // Estructura de la transición
      Trans17 : G7_TransitionPlus_V6;   // Estructura de la transición
      Trans18 : G7_TransitionPlus_V6;   // Estructura de la transición
      Trans19 : G7_TransitionPlus_V6;   // Estructura de la transición
      Trans20 : G7_TransitionPlus_V6;   // Estructura de la transición
      Trans21 : G7_TransitionPlus_V6;   // Estructura de la transición
      Trans22 : G7_TransitionPlus_V6;   // Estructura de la transición
      Trans23 : G7_TransitionPlus_V6;   // Estructura de la transición
      Trans24 : G7_TransitionPlus_V6;   // Estructura de la transición
      X40 : G7_StepPlus_V6;   // Estructura de la etapa
      X41 : G7_StepPlus_V6;   // Estructura de la etapa
      X42 : G7_StepPlus_V6;   // Estructura de la etapa
      X45 : G7_StepPlus_V6;   // Estructura de la etapa
      X43 : G7_StepPlus_V6;   // Estructura de la etapa
      X46 : G7_StepPlus_V6;   // Estructura de la etapa
      X47 : G7_StepPlus_V6;   // Estructura de la etapa
      X44 : G7_StepPlus_V6;   // Estructura de la etapa
      X52 : G7_StepPlus_V6;   // Estructura de la etapa
      X48 : G7_StepPlus_V6;   // Estructura de la etapa
      X49 : G7_StepPlus_V6;   // Estructura de la etapa
      X53 : G7_StepPlus_V6;   // Estructura de la etapa
      X54 : G7_StepPlus_V6;   // Estructura de la etapa
      X50 : G7_StepPlus_V6;   // Estructura de la etapa
      X51 : G7_StepPlus_V6;   // Estructura de la etapa
      X55 : G7_StepPlus_V6;   // Estructura de la etapa
      X56 : G7_StepPlus_V6;   // Estructura de la etapa
      X57 : G7_StepPlus_V6;   // Estructura de la etapa
      X58 : G7_StepPlus_V6;   // Estructura de la etapa
      SINI : Array[0..1] of USInt;
      LSTT : Array[0..22] of USInt;
      ATAJ : Array[0..22] of USInt;
      ATAB : Array[0..22] of USInt;
      PSTT : Array[0..22] of USInt;
      NSTT : Array[0..22] of USInt;
      ASSJ : Array[0..18] of USInt;
      ASSB : Array[0..18] of USInt;
      PTTS : Array[0..18] of USInt;
      NTTS : Array[0..18] of USInt;
      SW_SQTS : Array[0..18] of USInt;
      SWITCH : Array[0..7] of USInt;
      TVX : Array[0..8] of USInt;
      TTX : Array[0..8] of USInt;
      TSX : Array[0..1] of USInt;
      S00X : Array[0..1] of USInt;
      SOFFX : Array[0..1] of USInt;
      SONX : Array[0..1] of USInt;
      SAX : Array[0..1] of USInt;
      SERRX : Array[0..19] of USInt;
      SMX : Array[0..19] of USInt;
      S0X : Array[0..19] of USInt;
      S1X : Array[0..19] of USInt;
      IL_ALARM_INST : Diag_Alarm;
      SUP_ALARM_INST : Diag_Alarm;
      STEP_TIME_ALARM_INST : Diag_Alarm;
      IEC_TIMER_INST : IEC_TIMER;
      TRANSACTION_FLAG : Bool := false;
   END_VAR
   // SINI[0] := 2;
   // LSTT[0] := 255;
   // LSTT[1] := 255;
   // LSTT[2] := 255;
   // LSTT[3] := 255;
   // LSTT[4] := 255;
   // LSTT[5] := 255;
   // LSTT[6] := 255;
   // LSTT[7] := 255;
   // LSTT[8] := 255;
   // LSTT[9] := 255;
   // LSTT[10] := 255;
   // LSTT[11] := 255;
   // LSTT[12] := 255;
   // LSTT[13] := 255;
   // LSTT[14] := 255;
   // LSTT[15] := 255;
   // LSTT[16] := 255;
   // LSTT[17] := 255;
   // LSTT[18] := 255;
   // ATAJ[1] := 1;
   // ATAJ[2] := 2;
   // ATAJ[3] := 3;
   // ATAJ[4] := 4;
   // ATAJ[5] := 5;
   // ATAJ[6] := 6;
   // ATAJ[7] := 7;
   // ATAJ[8] := 8;
   // ATAJ[9] := 9;
   // ATAJ[10] := 10;
   // ATAJ[11] := 11;
   // ATAJ[12] := 12;
   // ATAJ[13] := 13;
   // ATAJ[14] := 14;
   // ATAJ[15] := 15;
   // ATAJ[16] := 16;
   // ATAJ[17] := 20;
   // ATAJ[18] := 21;
   // ATAJ[19] := 19;
   // ATAB[1] := 22;
   // ATAB[2] := 1;
   // ATAB[3] := 3;
   // ATAB[4] := 4;
   // ATAB[5] := 5;
   // ATAB[6] := 6;
   // ATAB[7] := 10;
   // ATAB[8] := 9;
   // ATAB[9] := 8;
   // ATAB[10] := 7;
   // ATAB[11] := 11;
   // ATAB[12] := 12;
   // ATAB[13] := 13;
   // ATAB[14] := 14;
   // ATAB[15] := 15;
   // ATAB[16] := 16;
   // ATAB[17] := 17;
   // ATAB[18] := 18;
   // ATAB[19] := 19;
   // PSTT[1] := 1;
   // PSTT[2] := 1;
   // PSTT[3] := 2;
   // PSTT[4] := 3;
   // PSTT[5] := 4;
   // PSTT[6] := 5;
   // PSTT[7] := 6;
   // PSTT[8] := 7;
   // PSTT[9] := 7;
   // PSTT[10] := 6;
   // PSTT[11] := 8;
   // PSTT[12] := 9;
   // PSTT[13] := 10;
   // PSTT[14] := 11;
   // PSTT[15] := 12;
   // PSTT[16] := 13;
   // PSTT[17] := 14;
   // PSTT[18] := 15;
   // PSTT[19] := 16;
   // NSTT[0] := 1;
   // NSTT[1] := 2;
   // NSTT[2] := 3;
   // NSTT[3] := 4;
   // NSTT[4] := 5;
   // NSTT[5] := 7;
   // NSTT[6] := 6;
   // NSTT[7] := 8;
   // NSTT[8] := 9;
   // NSTT[9] := 17;
   // NSTT[10] := 18;
   // NSTT[11] := 11;
   // NSTT[12] := 10;
   // NSTT[13] := 13;
   // NSTT[14] := 12;
   // NSTT[15] := 15;
   // NSTT[16] := 14;
   // NSTT[17] := 16;
   // NSTT[18] := 16;
   // ASSJ[1] := 1;
   // ASSJ[2] := 2;
   // ASSJ[3] := 3;
   // ASSJ[4] := 4;
   // ASSJ[5] := 5;
   // ASSJ[6] := 6;
   // ASSJ[7] := 7;
   // ASSJ[8] := 8;
   // ASSJ[9] := 9;
   // ASSJ[10] := 10;
   // ASSJ[11] := 11;
   // ASSJ[12] := 12;
   // ASSJ[13] := 13;
   // ASSJ[14] := 14;
   // ASSJ[15] := 15;
   // ASSJ[16] := 16;
   // ASSB[1] := 1;
   // ASSB[2] := 2;
   // ASSB[3] := 3;
   // ASSB[4] := 4;
   // ASSB[5] := 5;
   // ASSB[6] := 6;
   // ASSB[7] := 7;
   // ASSB[8] := 8;
   // ASSB[9] := 9;
   // ASSB[10] := 10;
   // ASSB[11] := 11;
   // ASSB[12] := 12;
   // ASSB[13] := 13;
   // ASSB[14] := 14;
   // ASSB[15] := 15;
   // ASSB[16] := 16;
   // PTTS[0] := 255;
   // PTTS[2] := 1;
   // PTTS[3] := 2;
   // PTTS[4] := 3;
   // PTTS[5] := 4;
   // PTTS[6] := 6;
   // PTTS[7] := 5;
   // PTTS[8] := 7;
   // PTTS[9] := 8;
   // PTTS[10] := 12;
   // PTTS[11] := 11;
   // PTTS[12] := 14;
   // PTTS[13] := 13;
   // PTTS[14] := 16;
   // PTTS[15] := 15;
   // PTTS[16] := 17;
   // NTTS[1] := 1;
   // NTTS[2] := 3;
   // NTTS[3] := 4;
   // NTTS[4] := 5;
   // NTTS[5] := 6;
   // NTTS[6] := 7;
   // NTTS[7] := 8;
   // NTTS[8] := 11;
   // NTTS[9] := 12;
   // NTTS[10] := 13;
   // NTTS[11] := 14;
   // NTTS[12] := 15;
   // NTTS[13] := 16;
   // NTTS[14] := 17;
   // NTTS[15] := 18;
   // NTTS[16] := 19;
   // SW_SQTS[2] := 1;
   // SW_SQTS[3] := 2;
   // SW_SQTS[4] := 1;
   // SW_SQTS[5] := 2;
   // SW_SQTS[6] := 2;
   // SW_SQTS[7] := 1;
   // SW_SQTS[8] := 3;
   // SW_SQTS[9] := 4;
   // SW_SQTS[10] := 4;
   // SW_SQTS[11] := 3;
   // SW_SQTS[12] := 3;
   // SW_SQTS[13] := 4;
   // SW_SQTS[14] := 4;
   // SW_SQTS[15] := 3;
   // SW_SQTS[16] := 5;
   // TVX[0] := 16#1;
   // TTX[0] := 16#1;
   // TSX[0] := 16#1;
   // S00X[0] := 16#1;
   // SOFFX[0] := 16#1;
   // SONX[0] := 16#1;
   // SAX[0] := 16#1;
   // SERRX[0] := 16#1;
   // SMX[0] := 16#1;
   // S0X[0] := 16#1;
   // S1X[0] := 16#1;
   // LSTT[20] := 255;
   // LSTT[21] := 255;
   // ATAJ[20] := 18;
   // ATAJ[21] := 17;
   // ATAB[20] := 20;
   // ATAB[21] := 21;
   // PSTT[20] := 17;
   // PSTT[21] := 18;
   // NSTT[20] := 16;
   // NSTT[21] := 16;
   // ASSJ[17] := 17;
   // ASSJ[18] := 18;
   // ASSB[17] := 17;
   // ASSB[18] := 18;
   // PTTS[17] := 9;
   // PTTS[18] := 10;
   // NTTS[17] := 20;
   // NTTS[18] := 21;
   // SW_SQTS[17] := 6;
   // SW_SQTS[18] := 7;
   // ATAJ[22] := 22;
   // ATAB[22] := 2;
   // PSTT[22] := 1;
BEGIN
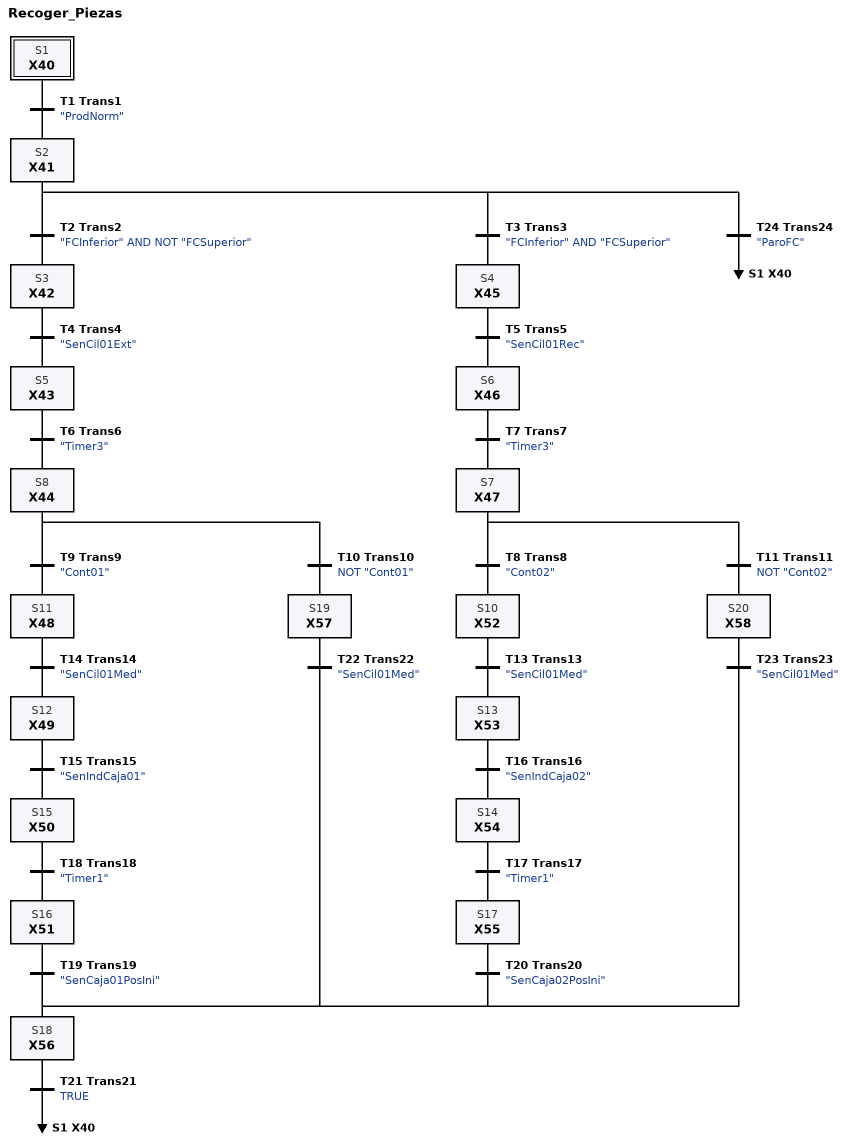
   // sequencer 1
   INITIAL_STEP X40:   // S1, max time T#10S, warning time T#7S
   END_STEP
   TRANSITION Trans1 FROM X40 TO X41   // T1
      := "ProdNorm";
   END_TRANSITION
   STEP X41:   // S2, max time T#10S, warning time T#7S
   END_STEP
   TRANSITION Trans2 FROM X41 TO X42   // T2
      := "FCInferior" AND NOT "FCSuperior";
   END_TRANSITION
   TRANSITION Trans3 FROM X41 TO X45   // T3
      := "FCInferior" AND "FCSuperior";
   END_TRANSITION
   TRANSITION Trans24 FROM X41 TO X40   // T24, jump
      := "ParoFC";
   END_TRANSITION
   STEP X42:   // S3, max time T#10S, warning time T#7S
   END_STEP
   TRANSITION Trans4 FROM X42 TO X43   // T4
      := "SenCil01Ext";
   END_TRANSITION
   STEP X45:   // S4, max time T#10S, warning time T#7S
   END_STEP
   TRANSITION Trans5 FROM X45 TO X46   // T5
      := "SenCil01Rec";
   END_TRANSITION
   STEP X43:   // S5, max time T#10S, warning time T#7S
   END_STEP
   TRANSITION Trans6 FROM X43 TO X44   // T6
      := "Timer3";
   END_TRANSITION
   STEP X46:   // S6, max time T#10S, warning time T#7S
   END_STEP
   TRANSITION Trans7 FROM X46 TO X47   // T7
      := "Timer3";
   END_TRANSITION
   STEP X47:   // S7, max time T#10S, warning time T#7S
   END_STEP
   TRANSITION Trans8 FROM X47 TO X52   // T8
      := "Cont02";
   END_TRANSITION
   TRANSITION Trans11 FROM X47 TO X58   // T11
      := NOT "Cont02";
   END_TRANSITION
   STEP X44:   // S8, max time T#10S, warning time T#7S
   END_STEP
   TRANSITION Trans9 FROM X44 TO X48   // T9
      := "Cont01";
   END_TRANSITION
   TRANSITION Trans10 FROM X44 TO X57   // T10
      := NOT "Cont01";
   END_TRANSITION
   STEP X48:   // S11, max time T#10S, warning time T#7S
   END_STEP
   TRANSITION Trans14 FROM X48 TO X49   // T14
      := "SenCil01Med";
   END_TRANSITION
   STEP X52:   // S10, max time T#10S, warning time T#7S
   END_STEP
   TRANSITION Trans13 FROM X52 TO X53   // T13
      := "SenCil01Med";
   END_TRANSITION
   STEP X49:   // S12, max time T#10S, warning time T#7S
   END_STEP
   TRANSITION Trans15 FROM X49 TO X50   // T15
      := "SenIndCaja01";
   END_TRANSITION
   STEP X53:   // S13, max time T#10S, warning time T#7S
   END_STEP
   TRANSITION Trans16 FROM X53 TO X54   // T16
      := "SenIndCaja02";
   END_TRANSITION
   STEP X54:   // S14, max time T#10S, warning time T#7S
   END_STEP
   TRANSITION Trans17 FROM X54 TO X55   // T17
      := "Timer1";
   END_TRANSITION
   STEP X50:   // S15, max time T#10S, warning time T#7S
   END_STEP
   TRANSITION Trans18 FROM X50 TO X51   // T18
      := "Timer1";
   END_TRANSITION
   STEP X51:   // S16, max time T#10S, warning time T#7S
   END_STEP
   TRANSITION Trans19 FROM X51 TO X56   // T19
      := "SenCaja01PosIni";
   END_TRANSITION
   STEP X55:   // S17, max time T#10S, warning time T#7S
   END_STEP
   TRANSITION Trans20 FROM X55 TO X56   // T20
      := "SenCaja02PosIni";
   END_TRANSITION
   STEP X56:   // S18, max time T#10S, warning time T#7S
   END_STEP
   TRANSITION Trans21 FROM X56 TO X40   // T21, jump
      := TRUE;
   END_TRANSITION
   STEP X57:   // S19, max time T#10S, warning time T#7S
   END_STEP
   TRANSITION Trans22 FROM X57 TO X56   // T22
      := "SenCil01Med";
   END_TRANSITION
   STEP X58:   // S20, max time T#10S, warning time T#7S
   END_STEP
   TRANSITION Trans23 FROM X58 TO X56   // T23
      := "SenCil01Med";
   END_TRANSITION
END_FUNCTION_BLOCK

FUNCTION_BLOCK "Marcha_Fin"   // FB7, GRAPH_PLUS
{ S7_Optimized_Access := 'TRUE' }
VERSION : 0.1
   VAR_INPUT
      OFF_SQ : Bool := false;   // Desactivar cadena
      INIT_SQ : Bool := false;   // Poner cadena en estado inicial
      ACK_EF : Bool := false;   // Acusar todos los errores y fallos
      S_PREV : Bool := false;   // Mostrar la etapa anterior en el parámetro S_NO
      S_NEXT : Bool := false;   // Mostrar la etapa siguiente en el parámetro S_NO
      SW_AUTO : Bool := false;   // Modo automático
      SW_TAP : Bool := false;   // Semiautomático/continuar con transición
      SW_TOP : Bool := false;   // Semiautomático/transición ignorada
      SW_MAN : Bool := false;   // Modo manual
      S_SEL : Int := 0;   // Seleccionar la etapa que debe mostrarse en S_NO
      S_ON : Bool := false;   // Activar la etapa del parámetro S_NO
      S_OFF : Bool := false;   // Desactivar el incremento presente en el parámetro S_NO
      T_PUSH : Bool := false;   // Habilitar conmutación de transición en modo semiautomático
   END_VAR
   VAR_OUTPUT
      S_NO : Int := 0;   // Número de etapa
      S_MORE : Bool := false;   // Existen más etapas que pueden mostrarse en S_NO.
      S_ACTIVE : Bool := false;   // El incremento presente en el parámetro S_NO está activo
      ERR_FLT : Bool := false;   // Error de grupo interlock o supervisión
      AUTO_ON : Bool := false;   // Modo automático activado
      TAP_ON : Bool := false;   // Modo semiautomático/etapa con transición activada
      TOP_ON : Bool := false;   // Modo semiautomático/Ignorar transición activado
      MAN_ON : Bool := false;   // Modo manual activado
   END_VAR
   VAR
      HMI_INFO : Array[0..11] of UInt;
      IF_PAR : G7_IfParPlus_V6;
      RT_DATA : G7_RTDataPlus_V6;   // Área de datos interna
      Trans1 : G7_TransitionPlus_V6;   // Estructura de la transición
      Trans2 : G7_TransitionPlus_V6;   // Estructura de la transición
      Trans3 : G7_TransitionPlus_V6;   // Estructura de la transición
      Trans4 : G7_TransitionPlus_V6;   // Estructura de la transición
      Trans5 : G7_TransitionPlus_V6;   // Estructura de la transición
      Trans6 : G7_TransitionPlus_V6;   // Estructura de la transición
      Trans8 : G7_TransitionPlus_V6;   // Estructura de la transición
      Trans9 : G7_TransitionPlus_V6;   // Estructura de la transición
      Trans10 : G7_TransitionPlus_V6;   // Estructura de la transición
      Trans11 : G7_TransitionPlus_V6;   // Estructura de la transición
      Trans12 : G7_TransitionPlus_V6;   // Estructura de la transición
      Trans13 : G7_TransitionPlus_V6;   // Estructura de la transición
      Trans15 : G7_TransitionPlus_V6;   // Estructura de la transición
      Trans16 : G7_TransitionPlus_V6;   // Estructura de la transición
      X80 : G7_StepPlus_V6;   // Estructura de la etapa
      X84 : G7_StepPlus_V6;   // Estructura de la etapa
      X82 : G7_StepPlus_V6;   // Estructura de la etapa
      X81 : G7_StepPlus_V6;   // Estructura de la etapa
      X83 : G7_StepPlus_V6;   // Estructura de la etapa
      X85 : G7_StepPlus_V6;   // Estructura de la etapa
      X87 : G7_StepPlus_V6;   // Estructura de la etapa
      X86 : G7_StepPlus_V6;   // Estructura de la etapa
      X89 : G7_StepPlus_V6;   // Estructura de la etapa
      X90 : G7_StepPlus_V6;   // Estructura de la etapa
      X91 : G7_StepPlus_V6;   // Estructura de la etapa
      X92 : G7_StepPlus_V6;   // Estructura de la etapa
      X88 : G7_StepPlus_V6;   // Estructura de la etapa
      X93 : G7_StepPlus_V6;   // Estructura de la etapa
      SINI : Array[0..4] of USInt;
      LSTT : Array[0..13] of USInt;
      ATAJ : Array[0..13] of USInt;
      ATAB : Array[0..13] of USInt;
      PSTT : Array[0..13] of USInt;
      NSTT : Array[0..13] of USInt;
      ASSJ : Array[0..13] of USInt;
      ASSB : Array[0..13] of USInt;
      PTTS : Array[0..13] of USInt;
      NTTS : Array[0..13] of USInt;
      SW_SQTS : Array[0..13] of USInt;
      SWITCH : Array[0..10] of USInt;
      TVX : Array[0..7] of USInt;
      TTX : Array[0..7] of USInt;
      TSX : Array[0..4] of USInt;
      S00X : Array[0..4] of USInt;
      SOFFX : Array[0..4] of USInt;
      SONX : Array[0..4] of USInt;
      SAX : Array[0..4] of USInt;
      SERRX : Array[0..14] of USInt;
      SMX : Array[0..14] of USInt;
      S0X : Array[0..14] of USInt;
      S1X : Array[0..14] of USInt;
      IL_ALARM_INST : Diag_Alarm;
      SUP_ALARM_INST : Diag_Alarm;
      STEP_TIME_ALARM_INST : Diag_Alarm;
      IEC_TIMER_INST : IEC_TIMER;
      TRANSACTION_FLAG : Bool := false;
   END_VAR
   // SINI[0] := 2;
   // SINI[2] := 255;
   // SINI[3] := 255;
   // SINI[4] := 255;
   // LSTT[0] := 255;
   // LSTT[1] := 255;
   // LSTT[2] := 255;
   // LSTT[3] := 255;
   // LSTT[4] := 255;
   // LSTT[5] := 255;
   // LSTT[6] := 255;
   // LSTT[7] := 255;
   // LSTT[8] := 255;
   // LSTT[9] := 255;
   // LSTT[10] := 255;
   // LSTT[11] := 255;
   // LSTT[13] := 255;
   // ATAJ[1] := 1;
   // ATAJ[2] := 2;
   // ATAJ[3] := 9;
   // ATAJ[4] := 4;
   // ATAJ[5] := 5;
   // ATAJ[6] := 7;
   // ATAJ[7] := 6;
   // ATAJ[8] := 8;
   // ATAJ[9] := 3;
   // ATAJ[10] := 10;
   // ATAJ[11] := 11;
   // ATAJ[12] := 12;
   // ATAJ[13] := 13;
   // ATAB[1] := 2;
   // ATAB[2] := 3;
   // ATAB[3] := 1;
   // ATAB[4] := 4;
   // ATAB[5] := 5;
   // ATAB[6] := 6;
   // ATAB[7] := 7;
   // ATAB[8] := 8;
   // ATAB[9] := 9;
   // ATAB[10] := 10;
   // ATAB[11] := 11;
   // ATAB[12] := 12;
   // ATAB[13] := 13;
   // PSTT[1] := 3;
   // PSTT[2] := 3;
   // PSTT[3] := 3;
   // PSTT[4] := 2;
   // PSTT[5] := 1;
   // PSTT[6] := 6;
   // PSTT[7] := 7;
   // PSTT[8] := 8;
   // PSTT[9] := 9;
   // PSTT[10] := 10;
   // PSTT[11] := 11;
   // PSTT[12] := 12;
   // PSTT[13] := 13;
   // NSTT[0] := 3;
   // NSTT[1] := 7;
   // NSTT[2] := 6;
   // NSTT[3] := 10;
   // NSTT[4] := 4;
   // NSTT[5] := 5;
   // NSTT[6] := 8;
   // NSTT[7] := 8;
   // NSTT[8] := 9;
   // NSTT[9] := 10;
   // NSTT[10] := 11;
   // NSTT[11] := 13;
   // NSTT[13] := 12;
   // ASSJ[1] := 1;
   // ASSJ[2] := 2;
   // ASSJ[3] := 3;
   // ASSJ[4] := 5;
   // ASSJ[5] := 13;
   // ASSJ[6] := 6;
   // ASSJ[7] := 7;
   // ASSJ[8] := 8;
   // ASSJ[9] := 9;
   // ASSJ[10] := 10;
   // ASSJ[11] := 11;
   // ASSJ[12] := 12;
   // ASSJ[13] := 4;
   // ASSB[1] := 3;
   // ASSB[2] := 1;
   // ASSB[3] := 2;
   // ASSB[4] := 4;
   // ASSB[5] := 5;
   // ASSB[6] := 6;
   // ASSB[7] := 7;
   // ASSB[8] := 8;
   // ASSB[9] := 9;
   // ASSB[10] := 10;
   // ASSB[11] := 11;
   // ASSB[12] := 12;
   // ASSB[13] := 13;
   // PTTS[0] := 255;
   // PTTS[4] := 4;
   // PTTS[5] := 5;
   // PTTS[6] := 2;
   // PTTS[7] := 1;
   // PTTS[8] := 7;
   // PTTS[9] := 8;
   // PTTS[10] := 9;
   // PTTS[11] := 10;
   // PTTS[12] := 13;
   // PTTS[13] := 11;
   // NTTS[1] := 5;
   // NTTS[2] := 4;
   // NTTS[3] := 1;
   // NTTS[4] := 13;
   // NTTS[5] := 13;
   // NTTS[6] := 6;
   // NTTS[7] := 7;
   // NTTS[8] := 8;
   // NTTS[9] := 9;
   // NTTS[10] := 10;
   // NTTS[11] := 11;
   // NTTS[12] := 12;
   // NTTS[13] := 13;
   // SW_SQTS[1] := 1;
   // SW_SQTS[2] := 2;
   // SW_SQTS[3] := 3;
   // SW_SQTS[4] := 2;
   // SW_SQTS[5] := 1;
   // SW_SQTS[6] := 4;
   // SW_SQTS[7] := 5;
   // SW_SQTS[8] := 6;
   // SW_SQTS[9] := 6;
   // SW_SQTS[10] := 7;
   // SW_SQTS[11] := 7;
   // SW_SQTS[12] := 8;
   // SW_SQTS[13] := 7;
   // SWITCH[1] := 248;
   // SWITCH[2] := 233;
   // SWITCH[3] := 51;
   // SWITCH[4] := 96;
   // SWITCH[5] := 192;
   // SWITCH[6] := 128;
   // SWITCH[7] := 1;
   // SWITCH[8] := 3;
   // TVX[0] := 16#1;
   // TTX[0] := 16#1;
   // TSX[0] := 16#1;
   // S00X[0] := 16#1;
   // SOFFX[0] := 16#1;
   // SONX[0] := 16#1;
   // SAX[0] := 16#1;
   // SERRX[0] := 16#1;
   // SMX[0] := 16#1;
   // S0X[0] := 16#1;
   // S1X[0] := 16#1;
BEGIN
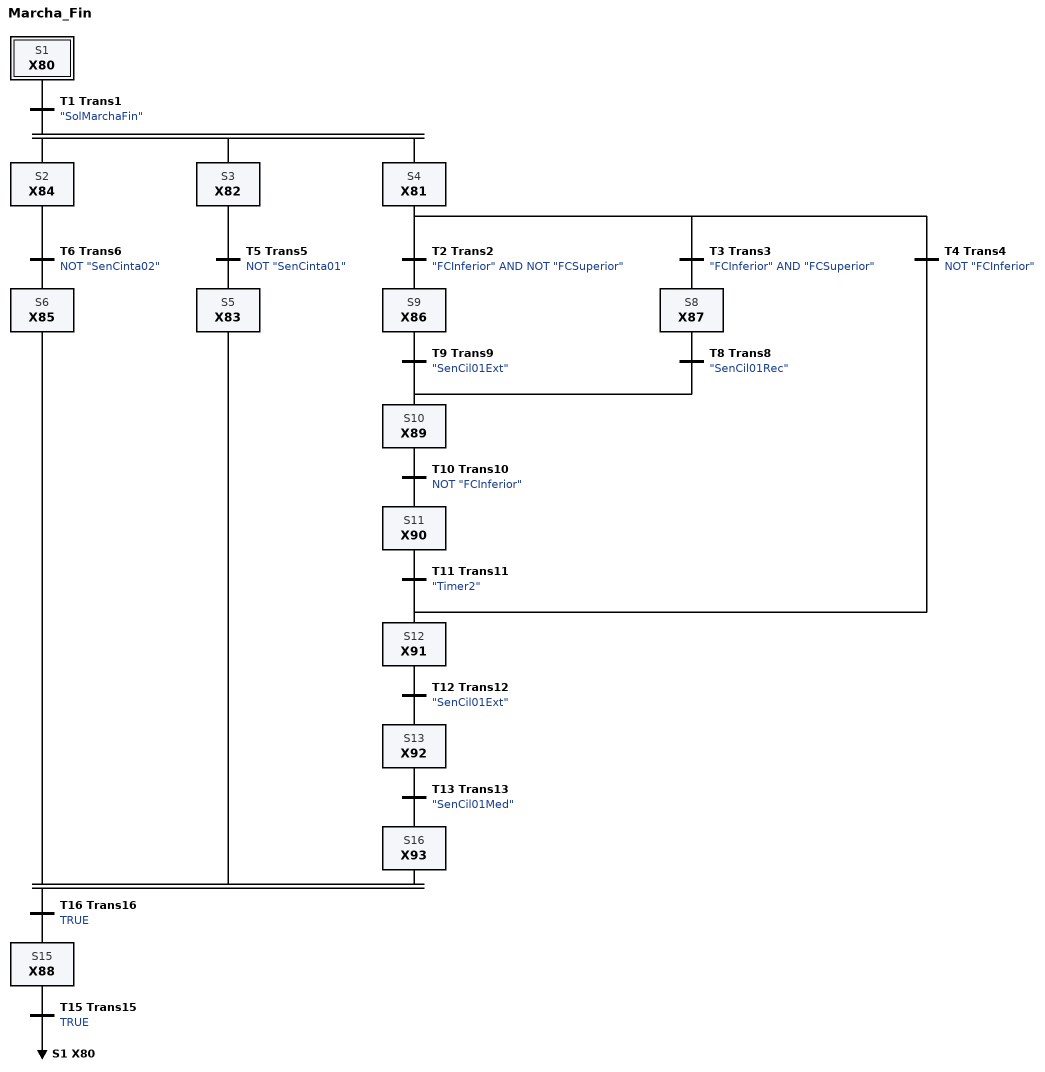
   // sequencer 1
   INITIAL_STEP X80:   // S1, max time T#10S, warning time T#7S
   END_STEP
   TRANSITION Trans1 FROM X80 TO (X84, X82, X81)   // T1
      := "SolMarchaFin";
   END_TRANSITION
   STEP X84:   // S2, max time T#10S, warning time T#7S
   END_STEP
   TRANSITION Trans6 FROM X84 TO X85   // T6
      := NOT "SenCinta02";
   END_TRANSITION
   STEP X82:   // S3, max time T#10S, warning time T#7S
   END_STEP
   TRANSITION Trans5 FROM X82 TO X83   // T5
      := NOT "SenCinta01";
   END_TRANSITION
   STEP X81:   // S4, max time T#10S, warning time T#7S
   END_STEP
   TRANSITION Trans2 FROM X81 TO X86   // T2
      := "FCInferior" AND NOT "FCSuperior";
   END_TRANSITION
   TRANSITION Trans3 FROM X81 TO X87   // T3
      := "FCInferior" AND "FCSuperior";
   END_TRANSITION
   TRANSITION Trans4 FROM X81 TO X91   // T4
      := NOT "FCInferior";
   END_TRANSITION
   STEP X83:   // S5, max time T#10S, warning time T#7S
   END_STEP
   TRANSITION Trans16 FROM (X85, X93, X83) TO X88   // T16
      := TRUE;
   END_TRANSITION
   STEP X85:   // S6, max time T#10S, warning time T#7S
   END_STEP
   STEP X89:   // S10, max time T#10S, warning time T#7S
   END_STEP
   TRANSITION Trans10 FROM X89 TO X90   // T10
      := NOT "FCInferior";
   END_TRANSITION
   STEP X87:   // S8, max time T#10S, warning time T#7S
   END_STEP
   TRANSITION Trans8 FROM X87 TO X89   // T8
      := "SenCil01Rec";
   END_TRANSITION
   STEP X86:   // S9, max time T#10S, warning time T#7S
   END_STEP
   TRANSITION Trans9 FROM X86 TO X89   // T9
      := "SenCil01Ext";
   END_TRANSITION
   STEP X90:   // S11, max time T#10S, warning time T#7S
   END_STEP
   TRANSITION Trans11 FROM X90 TO X91   // T11
      := "Timer2";
   END_TRANSITION
   STEP X91:   // S12, max time T#10S, warning time T#7S
   END_STEP
   TRANSITION Trans12 FROM X91 TO X92   // T12
      := "SenCil01Ext";
   END_TRANSITION
   STEP X92:   // S13, max time T#10S, warning time T#7S
   END_STEP
   TRANSITION Trans13 FROM X92 TO X93   // T13
      := "SenCil01Med";
   END_TRANSITION
   STEP X88:   // S15, max time T#10S, warning time T#7S
   END_STEP
   TRANSITION Trans15 FROM X88 TO X80   // T15, jump
      := TRUE;
   END_TRANSITION
   STEP X93:   // S16, max time T#10S, warning time T#7S
   END_STEP
END_FUNCTION_BLOCK

FUNCTION_BLOCK "Paro_Emergencia"   // FB8, GRAPH_PLUS
{ S7_Optimized_Access := 'TRUE' }
VERSION : 0.1
   VAR_INPUT
      OFF_SQ : Bool := false;   // Desactivar cadena
      INIT_SQ : Bool := false;   // Poner cadena en estado inicial
      ACK_EF : Bool := false;   // Acusar todos los errores y fallos
      S_PREV : Bool := false;   // Mostrar la etapa anterior en el parámetro S_NO
      S_NEXT : Bool := false;   // Mostrar la etapa siguiente en el parámetro S_NO
      SW_AUTO : Bool := false;   // Modo automático
      SW_TAP : Bool := false;   // Semiautomático/continuar con transición
      SW_TOP : Bool := false;   // Semiautomático/transición ignorada
      SW_MAN : Bool := false;   // Modo manual
      S_SEL : Int := 0;   // Seleccionar la etapa que debe mostrarse en S_NO
      S_ON : Bool := false;   // Activar la etapa del parámetro S_NO
      S_OFF : Bool := false;   // Desactivar el incremento presente en el parámetro S_NO
      T_PUSH : Bool := false;   // Habilitar conmutación de transición en modo semiautomático
   END_VAR
   VAR_OUTPUT
      S_NO : Int := 0;   // Número de etapa
      S_MORE : Bool := false;   // Existen más etapas que pueden mostrarse en S_NO.
      S_ACTIVE : Bool := false;   // El incremento presente en el parámetro S_NO está activo
      ERR_FLT : Bool := false;   // Error de grupo interlock o supervisión
      AUTO_ON : Bool := false;   // Modo automático activado
      TAP_ON : Bool := false;   // Modo semiautomático/etapa con transición activada
      TOP_ON : Bool := false;   // Modo semiautomático/Ignorar transición activado
      MAN_ON : Bool := false;   // Modo manual activado
   END_VAR
   VAR
      HMI_INFO : Array[0..11] of UInt;
      IF_PAR : G7_IfParPlus_V6;
      RT_DATA : G7_RTDataPlus_V6;   // Área de datos interna
      Trans1 : G7_TransitionPlus_V6;   // Estructura de la transición
      Trans3 : G7_TransitionPlus_V6;   // Estructura de la transición
      Trans5 : G7_TransitionPlus_V6;   // Estructura de la transición
      Trans6 : G7_TransitionPlus_V6;   // Estructura de la transición
      X300 : G7_StepPlus_V6;   // Estructura de la etapa
      X303 : G7_StepPlus_V6;   // Estructura de la etapa
      X301 : G7_StepPlus_V6;   // Estructura de la etapa
      X302 : G7_StepPlus_V6;   // Estructura de la etapa
      X304 : G7_StepPlus_V6;   // Estructura de la etapa
      X305 : G7_StepPlus_V6;   // Estructura de la etapa
      SINI : Array[0..4] of USInt;
      LSTT : Array[0..3] of USInt;
      ATAJ : Array[0..3] of USInt;
      ATAB : Array[0..3] of USInt;
      PSTT : Array[0..3] of USInt;
      NSTT : Array[0..3] of USInt;
      ASSJ : Array[0..5] of USInt;
      ASSB : Array[0..5] of USInt;
      PTTS : Array[0..5] of USInt;
      NTTS : Array[0..5] of USInt;
      SW_SQTS : Array[0..5] of USInt;
      SWITCH : Array[0..3] of USInt;
      TVX : Array[0..4] of USInt;
      TTX : Array[0..4] of USInt;
      TSX : Array[0..4] of USInt;
      S00X : Array[0..4] of USInt;
      SOFFX : Array[0..4] of USInt;
      SONX : Array[0..4] of USInt;
      SAX : Array[0..4] of USInt;
      SERRX : Array[0..6] of USInt;
      SMX : Array[0..6] of USInt;
      S0X : Array[0..6] of USInt;
      S1X : Array[0..6] of USInt;
      IL_ALARM_INST : Diag_Alarm;
      SUP_ALARM_INST : Diag_Alarm;
      STEP_TIME_ALARM_INST : Diag_Alarm;
      IEC_TIMER_INST : IEC_TIMER;
      TRANSACTION_FLAG : Bool := false;
   END_VAR
   // SINI[0] := 2;
   // SINI[2] := 255;
   // SINI[3] := 255;
   // LSTT[0] := 255;
   // LSTT[1] := 255;
   // LSTT[2] := 255;
   // ATAJ[1] := 1;
   // ATAJ[2] := 2;
   // ATAJ[3] := 3;
   // ATAB[1] := 1;
   // ATAB[2] := 2;
   // ATAB[3] := 3;
   // PSTT[1] := 2;
   // PSTT[2] := 3;
   // PSTT[3] := 4;
   // NSTT[0] := 2;
   // NSTT[1] := 3;
   // NSTT[2] := 4;
   // ASSJ[1] := 3;
   // ASSJ[2] := 2;
   // ASSJ[3] := 5;
   // ASSJ[4] := 4;
   // ASSB[1] := 2;
   // ASSB[2] := 5;
   // ASSB[3] := 3;
   // ASSB[4] := 4;
   // PTTS[0] := 255;
   // PTTS[3] := 1;
   // PTTS[4] := 2;
   // NTTS[1] := 2;
   // NTTS[2] := 1;
   // NTTS[3] := 2;
   // NTTS[4] := 3;
   // SW_SQTS[1] := 1;
   // SW_SQTS[2] := 2;
   // SW_SQTS[3] := 2;
   // SW_SQTS[4] := 3;
   // SWITCH[0] := 128;
   // SWITCH[1] := 74;
   // TVX[0] := 16#1;
   // TTX[0] := 16#1;
   // TSX[0] := 16#1;
   // S00X[0] := 16#1;
   // SOFFX[0] := 16#1;
   // SONX[0] := 16#1;
   // SAX[0] := 16#1;
   // SERRX[0] := 16#1;
   // SMX[0] := 16#1;
   // S0X[0] := 16#1;
   // S1X[0] := 16#1;
   // SINI[4] := 255;
   // ASSJ[5] := 1;
   // ASSB[5] := 1;
   // NTTS[5] := 2;
   // SW_SQTS[5] := 4;
   // SWITCH[2] := 96;
BEGIN
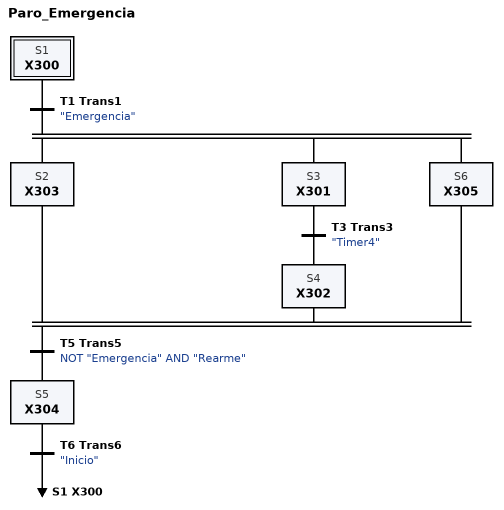
   // sequencer 1
   INITIAL_STEP X300:   // S1, max time T#10S, warning time T#7S
   END_STEP
   TRANSITION Trans1 FROM X300 TO (X303, X301, X305)   // T1
      := "Emergencia";
   END_TRANSITION
   STEP X303:   // S2, max time T#10S, warning time T#7S
   END_STEP
   STEP X301:   // S3, max time T#10S, warning time T#7S
   END_STEP
   TRANSITION Trans3 FROM X301 TO X302   // T3
      := "Timer4";
   END_TRANSITION
   STEP X302:   // S4, max time T#10S, warning time T#7S
   END_STEP
   STEP X304:   // S5, max time T#10S, warning time T#7S
   END_STEP
   TRANSITION Trans6 FROM X304 TO X300   // T6, jump
      := "Inicio";
   END_TRANSITION
   STEP X305:   // S6, max time T#10S, warning time T#7S
   END_STEP
   TRANSITION Trans5 FROM (X302, X303, X305) TO X304   // T5
      := NOT "Emergencia" AND "Rearme";
   END_TRANSITION
END_FUNCTION_BLOCK

ORGANIZATION_BLOCK "Main"   // OB1, LAD, ProgramCycle
TITLE = "Main Program Sweep (Cycle)"
{ S7_Optimized_Access := 'TRUE' }
VERSION : 0.1
   VAR_INPUT
      Initial_Call : Bool;   // Initial call of this OB
      Remanence : Bool;   // =True, if remanent data are available
   END_VAR
   VAR_TEMP   // added for the SCL form of the ladder/FBD networks
      _w1 : Bool;
      _w2 : Bool;
      _w3 : Bool;
   END_VAR
BEGIN

REGION Network 1: Bloques de Función
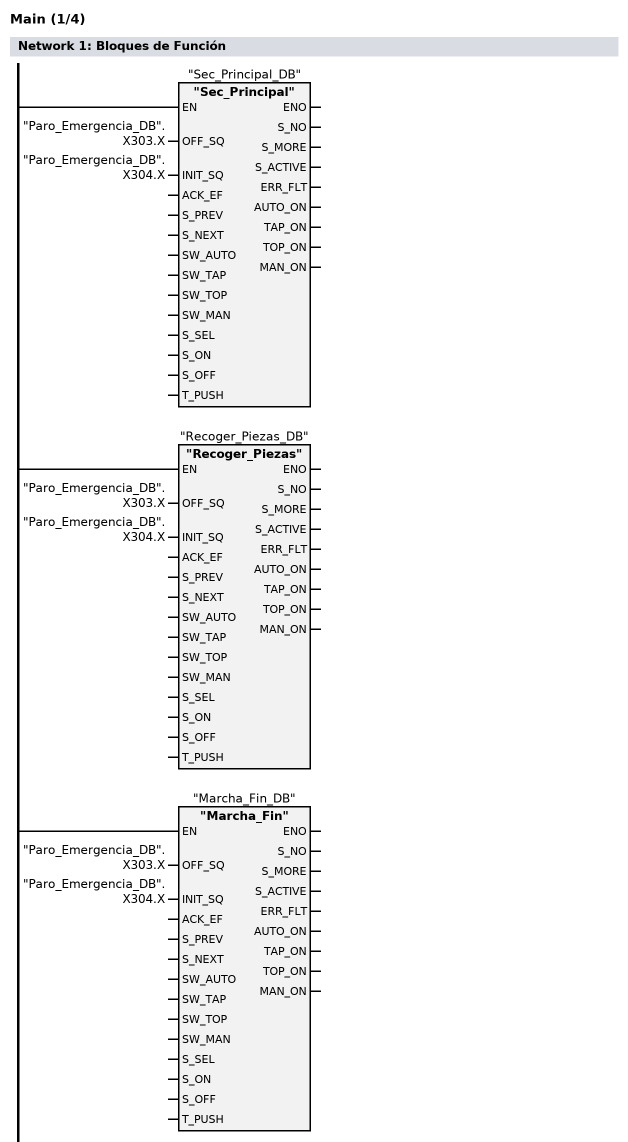
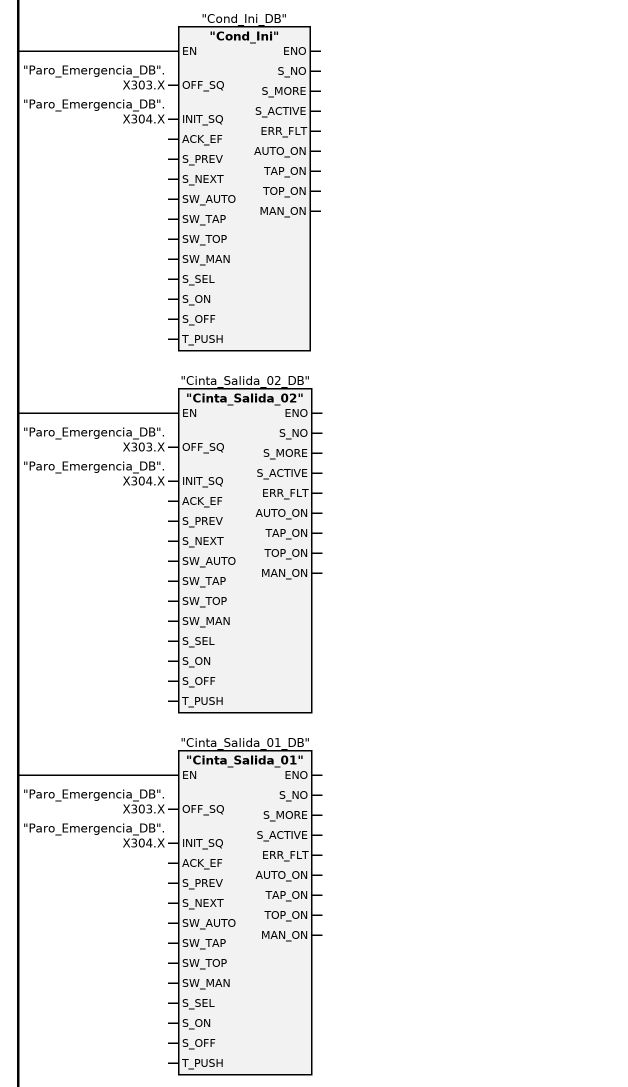
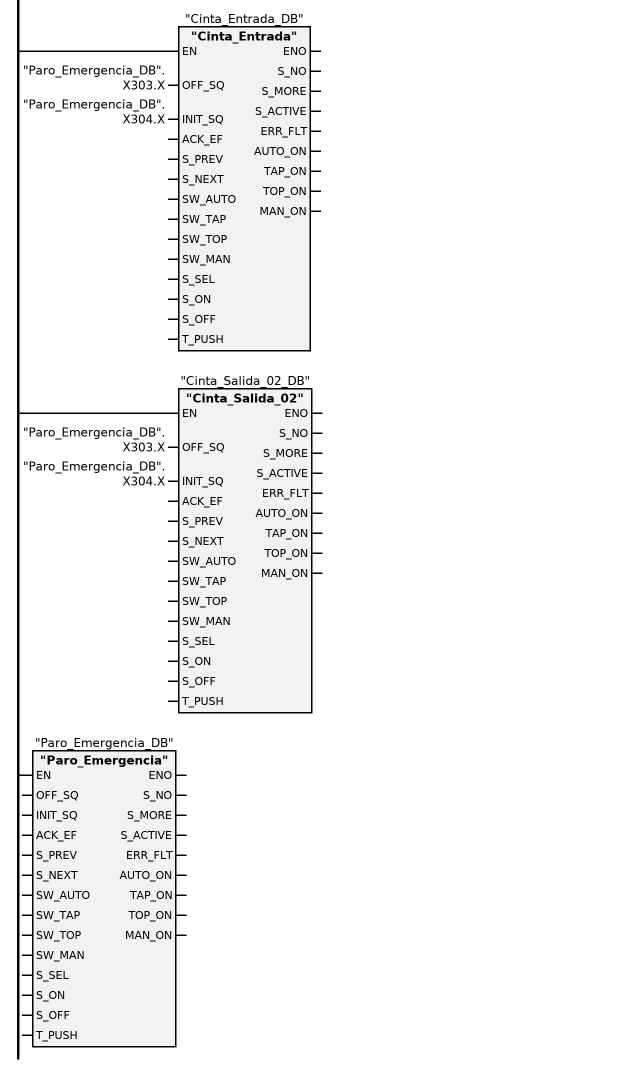
   RUNG wire#powerrail
      "Sec_Principal_DB"(OFF_SQ := "Paro_Emergencia_DB".X303.X, INIT_SQ := "Paro_Emergencia_DB".X304.X, ACK_EF :=, S_PREV :=, S_NEXT :=, SW_AUTO :=, SW_TAP :=, SW_TOP :=, SW_MAN :=, S_SEL :=, S_ON :=, S_OFF :=, T_PUSH :=, S_NO =>, S_MORE =>, S_ACTIVE =>, ERR_FLT =>, AUTO_ON =>, TAP_ON =>, TOP_ON =>, MAN_ON =>)
   END_RUNG
   RUNG wire#powerrail
      "Recoger_Piezas_DB"(OFF_SQ := "Paro_Emergencia_DB".X303.X, INIT_SQ := "Paro_Emergencia_DB".X304.X, ACK_EF :=, S_PREV :=, S_NEXT :=, SW_AUTO :=, SW_TAP :=, SW_TOP :=, SW_MAN :=, S_SEL :=, S_ON :=, S_OFF :=, T_PUSH :=, S_NO =>, S_MORE =>, S_ACTIVE =>, ERR_FLT =>, AUTO_ON =>, TAP_ON =>, TOP_ON =>, MAN_ON =>)
   END_RUNG
   RUNG wire#powerrail
      "Marcha_Fin_DB"(OFF_SQ := "Paro_Emergencia_DB".X303.X, INIT_SQ := "Paro_Emergencia_DB".X304.X, ACK_EF :=, S_PREV :=, S_NEXT :=, SW_AUTO :=, SW_TAP :=, SW_TOP :=, SW_MAN :=, S_SEL :=, S_ON :=, S_OFF :=, T_PUSH :=, S_NO =>, S_MORE =>, S_ACTIVE =>, ERR_FLT =>, AUTO_ON =>, TAP_ON =>, TOP_ON =>, MAN_ON =>)
   END_RUNG
   RUNG wire#powerrail
      "Cond_Ini_DB"(OFF_SQ := "Paro_Emergencia_DB".X303.X, INIT_SQ := "Paro_Emergencia_DB".X304.X, ACK_EF :=, S_PREV :=, S_NEXT :=, SW_AUTO :=, SW_TAP :=, SW_TOP :=, SW_MAN :=, S_SEL :=, S_ON :=, S_OFF :=, T_PUSH :=, S_NO =>, S_MORE =>, S_ACTIVE =>, ERR_FLT =>, AUTO_ON =>, TAP_ON =>, TOP_ON =>, MAN_ON =>)
   END_RUNG
   RUNG wire#powerrail
      "Cinta_Salida_02_DB"(OFF_SQ := "Paro_Emergencia_DB".X303.X, INIT_SQ := "Paro_Emergencia_DB".X304.X, ACK_EF :=, S_PREV :=, S_NEXT :=, SW_AUTO :=, SW_TAP :=, SW_TOP :=, SW_MAN :=, S_SEL :=, S_ON :=, S_OFF :=, T_PUSH :=, S_NO =>, S_MORE =>, S_ACTIVE =>, ERR_FLT =>, AUTO_ON =>, TAP_ON =>, TOP_ON =>, MAN_ON =>)
   END_RUNG
   RUNG wire#powerrail
      "Cinta_Salida_01_DB"(OFF_SQ := "Paro_Emergencia_DB".X303.X, INIT_SQ := "Paro_Emergencia_DB".X304.X, ACK_EF :=, S_PREV :=, S_NEXT :=, SW_AUTO :=, SW_TAP :=, SW_TOP :=, SW_MAN :=, S_SEL :=, S_ON :=, S_OFF :=, T_PUSH :=, S_NO =>, S_MORE =>, S_ACTIVE =>, ERR_FLT =>, AUTO_ON =>, TAP_ON =>, TOP_ON =>, MAN_ON =>)
   END_RUNG
   RUNG wire#powerrail
      "Cinta_Entrada_DB"(OFF_SQ := "Paro_Emergencia_DB".X303.X, INIT_SQ := "Paro_Emergencia_DB".X304.X, ACK_EF :=, S_PREV :=, S_NEXT :=, SW_AUTO :=, SW_TAP :=, SW_TOP :=, SW_MAN :=, S_SEL :=, S_ON :=, S_OFF :=, T_PUSH :=, S_NO =>, S_MORE =>, S_ACTIVE =>, ERR_FLT =>, AUTO_ON =>, TAP_ON =>, TOP_ON =>, MAN_ON =>)
   END_RUNG
   RUNG wire#powerrail
      "Cinta_Salida_02_DB"(OFF_SQ := "Paro_Emergencia_DB".X303.X, INIT_SQ := "Paro_Emergencia_DB".X304.X, ACK_EF :=, S_PREV :=, S_NEXT :=, SW_AUTO :=, SW_TAP :=, SW_TOP :=, SW_MAN :=, S_SEL :=, S_ON :=, S_OFF :=, T_PUSH :=, S_NO =>, S_MORE =>, S_ACTIVE =>, ERR_FLT =>, AUTO_ON =>, TAP_ON =>, TOP_ON =>, MAN_ON =>)
   END_RUNG
   RUNG wire#powerrail
      "Paro_Emergencia_DB"(OFF_SQ :=, INIT_SQ :=, ACK_EF :=, S_PREV :=, S_NEXT :=, SW_AUTO :=, SW_TAP :=, SW_TOP :=, SW_MAN :=, S_SEL :=, S_ON :=, S_OFF :=, T_PUSH :=, S_NO =>, S_MORE =>, S_ACTIVE =>, ERR_FLT =>, AUTO_ON =>, TAP_ON =>, TOP_ON =>, MAN_ON =>)
   END_RUNG
   // the same network as SCL:
   "Sec_Principal_DB"(OFF_SQ := "Paro_Emergencia_DB".X303.X, INIT_SQ := "Paro_Emergencia_DB".X304.X);   // "Sec_Principal"
   "Recoger_Piezas_DB"(OFF_SQ := "Paro_Emergencia_DB".X303.X, INIT_SQ := "Paro_Emergencia_DB".X304.X);   // "Recoger_Piezas"
   "Marcha_Fin_DB"(OFF_SQ := "Paro_Emergencia_DB".X303.X, INIT_SQ := "Paro_Emergencia_DB".X304.X);   // "Marcha_Fin"
   "Cond_Ini_DB"(OFF_SQ := "Paro_Emergencia_DB".X303.X, INIT_SQ := "Paro_Emergencia_DB".X304.X);   // "Cond_Ini"
   "Cinta_Salida_02_DB"(OFF_SQ := "Paro_Emergencia_DB".X303.X, INIT_SQ := "Paro_Emergencia_DB".X304.X);   // "Cinta_Salida_02"
   "Cinta_Salida_01_DB"(OFF_SQ := "Paro_Emergencia_DB".X303.X, INIT_SQ := "Paro_Emergencia_DB".X304.X);   // "Cinta_Salida_01"
   "Cinta_Entrada_DB"(OFF_SQ := "Paro_Emergencia_DB".X303.X, INIT_SQ := "Paro_Emergencia_DB".X304.X);   // "Cinta_Entrada"
   "Cinta_Salida_02_DB"(OFF_SQ := "Paro_Emergencia_DB".X303.X, INIT_SQ := "Paro_Emergencia_DB".X304.X);   // "Cinta_Salida_02"
   "Paro_Emergencia_DB"();   // "Paro_Emergencia"
END_REGION

REGION Network 2: Contadores y Temporizadores
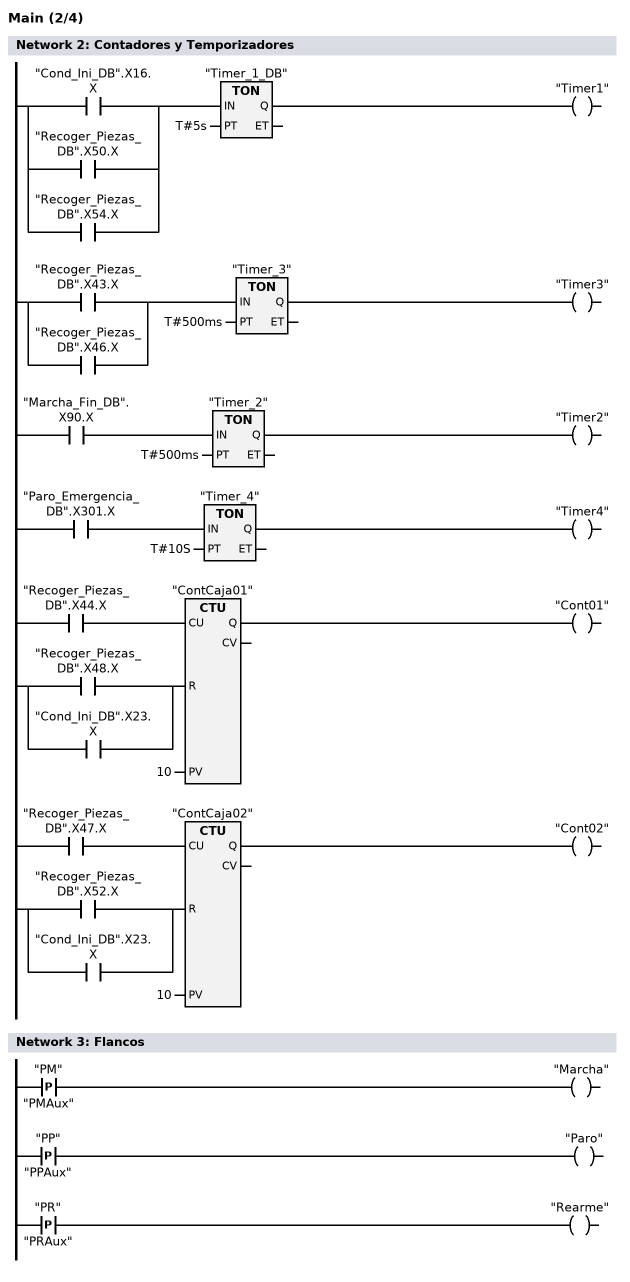
   "Timer_1_DB".TON(IN := "Cond_Ini_DB".X16.X OR "Recoger_Piezas_DB".X50.X OR "Recoger_Piezas_DB".X54.X,
                    PT := T#5s);
   "Timer1" := "Timer_1_DB".Q;
   "Timer_3".TON(IN := "Recoger_Piezas_DB".X43.X OR "Recoger_Piezas_DB".X46.X, PT := T#500ms);
   "Timer3" := "Timer_3".Q;
   "Timer_2".TON(IN := "Marcha_Fin_DB".X90.X, PT := T#500ms);
   "Timer2" := "Timer_2".Q;
   "Timer_4".TON(IN := "Paro_Emergencia_DB".X301.X, PT := T#10S);
   "Timer4" := "Timer_4".Q;
   "ContCaja01".CTU(CU := "Recoger_Piezas_DB".X44.X,
                    R := "Recoger_Piezas_DB".X48.X OR "Cond_Ini_DB".X23.X,
                    PV := 10);
   "Cont01" := "ContCaja01".Q;
   "ContCaja02".CTU(CU := "Recoger_Piezas_DB".X47.X,
                    R := "Recoger_Piezas_DB".X52.X OR "Cond_Ini_DB".X23.X,
                    PV := 10);
   "Cont02" := "ContCaja02".Q;
END_REGION

REGION Network 3: Flancos
   RUNG wire#powerrail
      P_Contact(operand := "PM", bit := "PMAux")
      Coil( "Marcha" )
   END_RUNG
   RUNG wire#powerrail
      P_Contact(operand := "PP", bit := "PPAux")
      Coil( "Paro" )
   END_RUNG
   RUNG wire#powerrail
      P_Contact(operand := "PR", bit := "PRAux")
      Coil( "Rearme" )
   END_RUNG
   // the same network as SCL:
   #_w1 := "PM" AND NOT "PMAux";   // rising edge of "PM"
   "PMAux" := "PM";
   "Marcha" := #_w1;
   #_w2 := "PP" AND NOT "PPAux";   // rising edge of "PP"
   "PPAux" := "PP";
   "Paro" := #_w2;
   #_w3 := "PR" AND NOT "PRAux";   // rising edge of "PR"
   "PRAux" := "PR";
   "Rearme" := #_w3;
END_REGION

REGION Network 4: Señales de Control
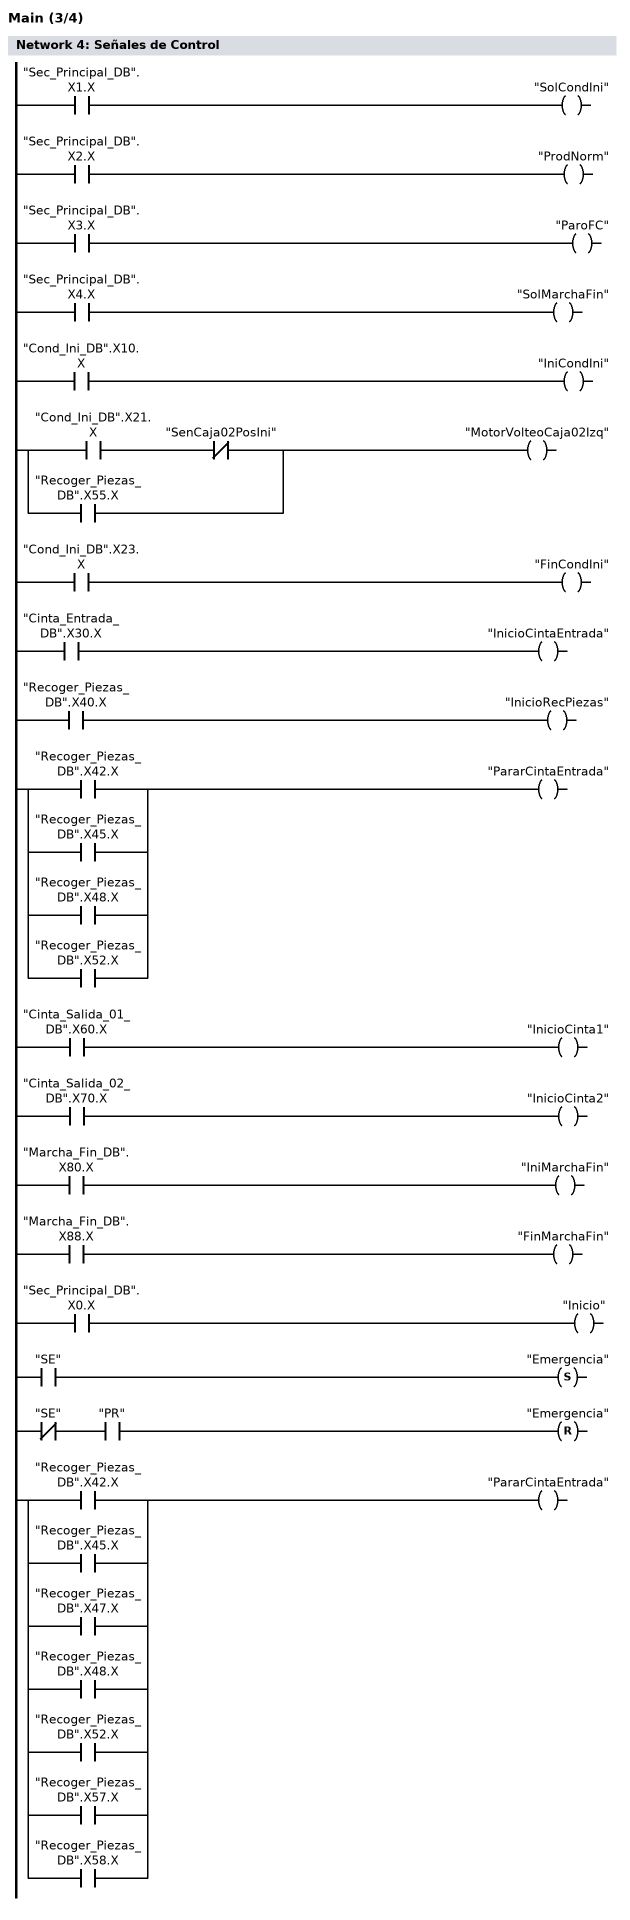
   RUNG wire#powerrail
      Contact( "Sec_Principal_DB".X1.X )
      Coil( "SolCondIni" )
   END_RUNG
   RUNG wire#powerrail
      Contact( "Sec_Principal_DB".X2.X )
      Coil( "ProdNorm" )
   END_RUNG
   RUNG wire#powerrail
      Contact( "Sec_Principal_DB".X3.X )
      Coil( "ParoFC" )
   END_RUNG
   RUNG wire#powerrail
      Contact( "Sec_Principal_DB".X4.X )
      Coil( "SolMarchaFin" )
   END_RUNG
   RUNG wire#powerrail
      Contact( "Cond_Ini_DB".X10.X )
      Coil( "IniCondIni" )
   END_RUNG
   RUNG wire#powerrail
      Contact( "Cond_Ini_DB".X21.X )
      I_Contact( "SenCaja02PosIni" )
      wire#w1
      Coil( "MotorVolteoCaja02Izq" )
   END_RUNG
   RUNG wire#powerrail
      Contact( "Recoger_Piezas_DB".X55.X )
   END_RUNG wire#w1
   RUNG wire#powerrail
      Contact( "Cond_Ini_DB".X23.X )
      Coil( "FinCondIni" )
   END_RUNG
   RUNG wire#powerrail
      Contact( "Cinta_Entrada_DB".X30.X )
      Coil( "InicioCintaEntrada" )
   END_RUNG
   RUNG wire#powerrail
      Contact( "Recoger_Piezas_DB".X40.X )
      Coil( "InicioRecPiezas" )
   END_RUNG
   RUNG wire#powerrail
      Contact( "Recoger_Piezas_DB".X42.X )
      wire#w2
      Coil( "PararCintaEntrada" )
   END_RUNG
   RUNG wire#powerrail
      Contact( "Recoger_Piezas_DB".X45.X )
   END_RUNG wire#w2
   RUNG wire#powerrail
      Contact( "Recoger_Piezas_DB".X48.X )
   END_RUNG wire#w2
   RUNG wire#powerrail
      Contact( "Recoger_Piezas_DB".X52.X )
   END_RUNG wire#w2
   RUNG wire#powerrail
      Contact( "Cinta_Salida_01_DB".X60.X )
      Coil( "InicioCinta1" )
   END_RUNG
   RUNG wire#powerrail
      Contact( "Cinta_Salida_02_DB".X70.X )
      Coil( "InicioCinta2" )
   END_RUNG
   RUNG wire#powerrail
      Contact( "Marcha_Fin_DB".X80.X )
      Coil( "IniMarchaFin" )
   END_RUNG
   RUNG wire#powerrail
      Contact( "Marcha_Fin_DB".X88.X )
      Coil( "FinMarchaFin" )
   END_RUNG
   RUNG wire#powerrail
      Contact( "Sec_Principal_DB".X0.X )
      Coil( "Inicio" )
   END_RUNG
   RUNG wire#powerrail
      Contact( "SE" )
      S_Coil( "Emergencia" )
   END_RUNG
   RUNG wire#powerrail
      I_Contact( "SE" )
      Contact( "PR" )
      R_Coil( "Emergencia" )
   END_RUNG
   RUNG wire#powerrail
      Contact( "Recoger_Piezas_DB".X42.X )
      wire#w3
      Coil( "PararCintaEntrada" )
   END_RUNG
   RUNG wire#powerrail
      Contact( "Recoger_Piezas_DB".X45.X )
   END_RUNG wire#w3
   RUNG wire#powerrail
      Contact( "Recoger_Piezas_DB".X47.X )
   END_RUNG wire#w3
   RUNG wire#powerrail
      Contact( "Recoger_Piezas_DB".X48.X )
   END_RUNG wire#w3
   RUNG wire#powerrail
      Contact( "Recoger_Piezas_DB".X52.X )
   END_RUNG wire#w3
   RUNG wire#powerrail
      Contact( "Recoger_Piezas_DB".X57.X )
   END_RUNG wire#w3
   RUNG wire#powerrail
      Contact( "Recoger_Piezas_DB".X58.X )
   END_RUNG wire#w3
   // the same network as SCL:
   "SolCondIni" := "Sec_Principal_DB".X1.X;
   "ProdNorm" := "Sec_Principal_DB".X2.X;
   "ParoFC" := "Sec_Principal_DB".X3.X;
   "SolMarchaFin" := "Sec_Principal_DB".X4.X;
   "IniCondIni" := "Cond_Ini_DB".X10.X;
   "MotorVolteoCaja02Izq" := ("Cond_Ini_DB".X21.X AND NOT "SenCaja02PosIni") OR "Recoger_Piezas_DB".X55.X;
   "FinCondIni" := "Cond_Ini_DB".X23.X;
   "InicioCintaEntrada" := "Cinta_Entrada_DB".X30.X;
   "InicioRecPiezas" := "Recoger_Piezas_DB".X40.X;
   "PararCintaEntrada" := "Recoger_Piezas_DB".X42.X OR "Recoger_Piezas_DB".X45.X OR "Recoger_Piezas_DB".X48.X OR "Recoger_Piezas_DB".X52.X;
   "InicioCinta1" := "Cinta_Salida_01_DB".X60.X;
   "InicioCinta2" := "Cinta_Salida_02_DB".X70.X;
   "IniMarchaFin" := "Marcha_Fin_DB".X80.X;
   "FinMarchaFin" := "Marcha_Fin_DB".X88.X;
   "Inicio" := "Sec_Principal_DB".X0.X;
   IF "SE" THEN "Emergencia" := TRUE; END_IF;
   IF NOT "SE" AND "PR" THEN "Emergencia" := FALSE; END_IF;
   "PararCintaEntrada" := "Recoger_Piezas_DB".X42.X OR "Recoger_Piezas_DB".X45.X OR "Recoger_Piezas_DB".X47.X OR "Recoger_Piezas_DB".X48.X OR "Recoger_Piezas_DB".X52.X OR "Recoger_Piezas_DB".X57.X OR "Recoger_Piezas_DB".X58.X;
END_REGION

REGION Network 5: Salidas del Programa
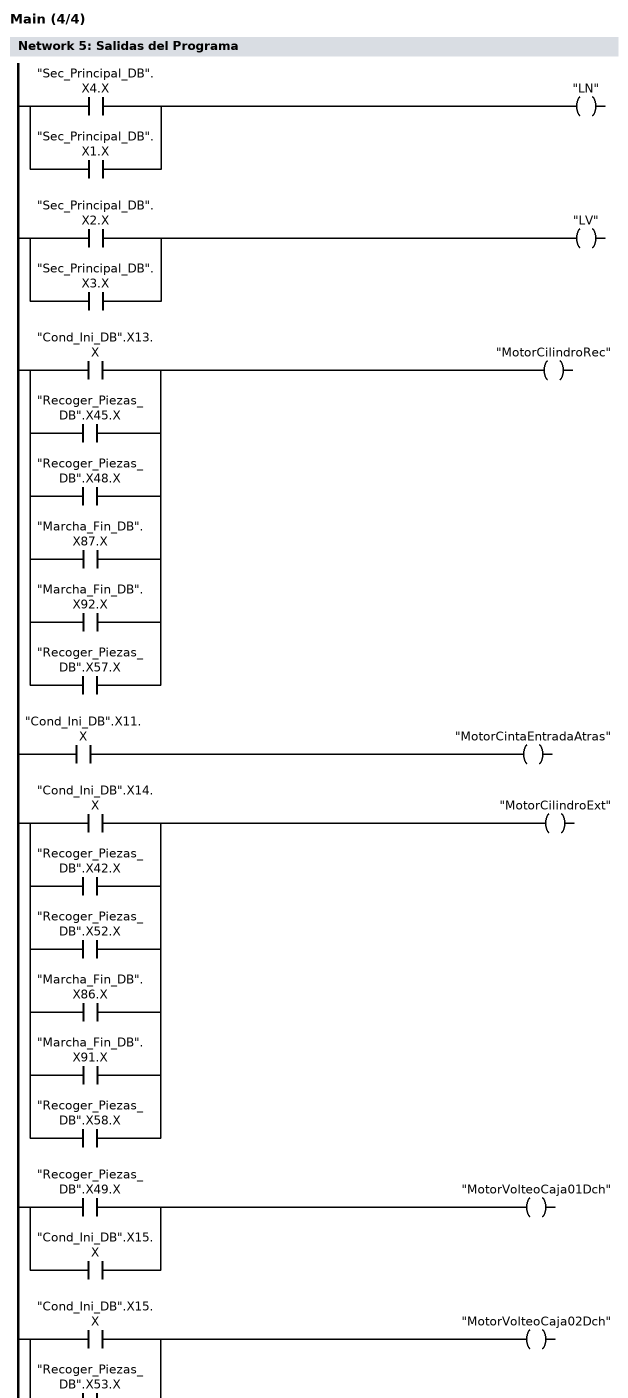
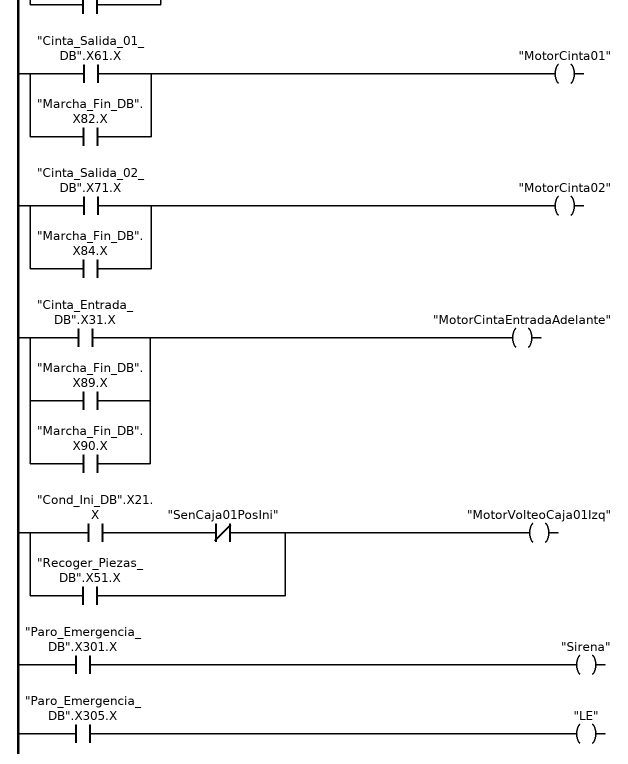
   RUNG wire#powerrail
      Contact( "Sec_Principal_DB".X4.X )
      wire#w1
      Coil( "LN" )
   END_RUNG
   RUNG wire#powerrail
      Contact( "Sec_Principal_DB".X1.X )
   END_RUNG wire#w1
   RUNG wire#powerrail
      Contact( "Sec_Principal_DB".X2.X )
      wire#w2
      Coil( "LV" )
   END_RUNG
   RUNG wire#powerrail
      Contact( "Sec_Principal_DB".X3.X )
   END_RUNG wire#w2
   RUNG wire#powerrail
      Contact( "Cond_Ini_DB".X13.X )
      wire#w3
      Coil( "MotorCilindroRec" )
   END_RUNG
   RUNG wire#powerrail
      Contact( "Recoger_Piezas_DB".X45.X )
   END_RUNG wire#w3
   RUNG wire#powerrail
      Contact( "Recoger_Piezas_DB".X48.X )
   END_RUNG wire#w3
   RUNG wire#powerrail
      Contact( "Marcha_Fin_DB".X87.X )
   END_RUNG wire#w3
   RUNG wire#powerrail
      Contact( "Marcha_Fin_DB".X92.X )
   END_RUNG wire#w3
   RUNG wire#powerrail
      Contact( "Recoger_Piezas_DB".X57.X )
   END_RUNG wire#w3
   RUNG wire#powerrail
      Contact( "Cond_Ini_DB".X11.X )
      Coil( "MotorCintaEntradaAtras" )
   END_RUNG
   RUNG wire#powerrail
      Contact( "Cond_Ini_DB".X14.X )
      wire#w4
      Coil( "MotorCilindroExt" )
   END_RUNG
   RUNG wire#powerrail
      Contact( "Recoger_Piezas_DB".X42.X )
   END_RUNG wire#w4
   RUNG wire#powerrail
      Contact( "Recoger_Piezas_DB".X52.X )
   END_RUNG wire#w4
   RUNG wire#powerrail
      Contact( "Marcha_Fin_DB".X86.X )
   END_RUNG wire#w4
   RUNG wire#powerrail
      Contact( "Marcha_Fin_DB".X91.X )
   END_RUNG wire#w4
   RUNG wire#powerrail
      Contact( "Recoger_Piezas_DB".X58.X )
   END_RUNG wire#w4
   RUNG wire#powerrail
      Contact( "Recoger_Piezas_DB".X49.X )
      wire#w5
      Coil( "MotorVolteoCaja01Dch" )
   END_RUNG
   RUNG wire#powerrail
      Contact( "Cond_Ini_DB".X15.X )
   END_RUNG wire#w5
   RUNG wire#powerrail
      Contact( "Cond_Ini_DB".X15.X )
      wire#w6
      Coil( "MotorVolteoCaja02Dch" )
   END_RUNG
   RUNG wire#powerrail
      Contact( "Recoger_Piezas_DB".X53.X )
   END_RUNG wire#w6
   RUNG wire#powerrail
      Contact( "Cinta_Salida_01_DB".X61.X )
      wire#w7
      Coil( "MotorCinta01" )
   END_RUNG
   RUNG wire#powerrail
      Contact( "Marcha_Fin_DB".X82.X )
   END_RUNG wire#w7
   RUNG wire#powerrail
      Contact( "Cinta_Salida_02_DB".X71.X )
      wire#w8
      Coil( "MotorCinta02" )
   END_RUNG
   RUNG wire#powerrail
      Contact( "Marcha_Fin_DB".X84.X )
   END_RUNG wire#w8
   RUNG wire#powerrail
      Contact( "Cinta_Entrada_DB".X31.X )
      wire#w9
      Coil( "MotorCintaEntradaAdelante" )
   END_RUNG
   RUNG wire#powerrail
      Contact( "Marcha_Fin_DB".X89.X )
   END_RUNG wire#w9
   RUNG wire#powerrail
      Contact( "Marcha_Fin_DB".X90.X )
   END_RUNG wire#w9
   RUNG wire#powerrail
      Contact( "Cond_Ini_DB".X21.X )
      I_Contact( "SenCaja01PosIni" )
      wire#w10
      Coil( "MotorVolteoCaja01Izq" )
   END_RUNG
   RUNG wire#powerrail
      Contact( "Recoger_Piezas_DB".X51.X )
   END_RUNG wire#w10
   RUNG wire#powerrail
      Contact( "Paro_Emergencia_DB".X301.X )
      Coil( "Sirena" )
   END_RUNG
   RUNG wire#powerrail
      Contact( "Paro_Emergencia_DB".X305.X )
      Coil( "LE" )
   END_RUNG
   // the same network as SCL:
   "LN" := "Sec_Principal_DB".X4.X OR "Sec_Principal_DB".X1.X;
   "LV" := "Sec_Principal_DB".X2.X OR "Sec_Principal_DB".X3.X;
   "MotorCilindroRec" := "Cond_Ini_DB".X13.X OR "Recoger_Piezas_DB".X45.X OR "Recoger_Piezas_DB".X48.X OR "Marcha_Fin_DB".X87.X OR "Marcha_Fin_DB".X92.X OR "Recoger_Piezas_DB".X57.X;
   "MotorCintaEntradaAtras" := "Cond_Ini_DB".X11.X;
   "MotorCilindroExt" := "Cond_Ini_DB".X14.X OR "Recoger_Piezas_DB".X42.X OR "Recoger_Piezas_DB".X52.X OR "Marcha_Fin_DB".X86.X OR "Marcha_Fin_DB".X91.X OR "Recoger_Piezas_DB".X58.X;
   "MotorVolteoCaja01Dch" := "Recoger_Piezas_DB".X49.X OR "Cond_Ini_DB".X15.X;
   "MotorVolteoCaja02Dch" := "Cond_Ini_DB".X15.X OR "Recoger_Piezas_DB".X53.X;
   "MotorCinta01" := "Cinta_Salida_01_DB".X61.X OR "Marcha_Fin_DB".X82.X;
   "MotorCinta02" := "Cinta_Salida_02_DB".X71.X OR "Marcha_Fin_DB".X84.X;
   "MotorCintaEntradaAdelante" := "Cinta_Entrada_DB".X31.X OR "Marcha_Fin_DB".X89.X OR "Marcha_Fin_DB".X90.X;
   "MotorVolteoCaja01Izq" := ("Cond_Ini_DB".X21.X AND NOT "SenCaja01PosIni") OR "Recoger_Piezas_DB".X51.X;
   "Sirena" := "Paro_Emergencia_DB".X301.X;
   "LE" := "Paro_Emergencia_DB".X305.X;
END_REGION
END_ORGANIZATION_BLOCK

(* ===== HMI "HMI_RT_2" =====
system functions are stored by id; their names below are inferred from use
connection "HMI_Conexión_2": ETHERNET, SMART_S7_1500_OMS

HMI tags "Tabla de variables estándar"
   "Número_imagen_variable" : UInt, internal
   "PM" : Bool = PLC PM AT %M0.0, 1 s
   "PP" : Bool = PLC PP AT %M0.1, 1 s
   "SE" : Bool = PLC SE AT %M0.2, 1 s
   "PR" : Bool = PLC PR AT %M0.3, 1 s
   "FCSuperior" : Bool = PLC FCSuperior AT %M0.4, 1 s
   "FCInferior" : Bool = PLC FCInferior AT %M0.5, 1 s
   "SenCintaEntrada" : Bool = PLC SenCintaEntrada AT %M0.6, 1 s
   "SenCaja01PosIni" : Bool = PLC SenCaja01PosIni AT %M0.7, 1 s
   "SenCaja02PosIni" : Bool = PLC SenCaja02PosIni AT %M1.0, 1 s
   "SenCil01Rec" : Bool = PLC SenCil01Rec AT %M1.1, 1 s
   "SenCil01Med" : Bool = PLC SenCil01Med AT %M1.2, 1 s
   "SenCil01Ext" : Bool = PLC SenCil01Ext AT %M1.3, 1 s
   "SenIndCaja01" : Bool = PLC SenIndCaja01 AT %M1.4, 1 s
   "SenIndCaja02" : Bool = PLC SenIndCaja02 AT %M1.5, 1 s
   "SenCinta01" : Bool = PLC SenCinta01 AT %M1.6, 1 s
   "SenCinta02" : Bool = PLC SenCinta02 AT %M1.7, 1 s
   "PMAux" : Bool = PLC PMAux AT %M2.0, 1 s
   "PPAux" : Bool = PLC PPAux AT %M2.1, 1 s
   "PRAux" : Bool = PLC PRAux AT %M2.2, 1 s
   "Marcha" : Bool = PLC Marcha AT %M4.4, 1 s
   "Paro" : Bool = PLC Paro AT %M4.5, 1 s
   "Rearme" : Bool = PLC Rearme AT %M4.6, 1 s
   "Inicio" : Bool = PLC Inicio AT %M2.4, 1 s
   "SolCondIni" : Bool = PLC SolCondIni AT %M2.5, 1 s
   "IniCondIni" : Bool = PLC IniCondIni AT %M2.6, 1 s
   "FinCondIni" : Bool = PLC FinCondIni AT %M2.7, 1 s
   "ProdNorm" : Bool = PLC ProdNorm AT %M3.0, 1 s
   "ParoFC" : Bool = PLC ParoFC AT %M3.1, 1 s
   "InicioCintaEntrada" : Bool = PLC InicioCintaEntrada AT %M3.2, 1 s
   "InicioRecPiezas" : Bool = PLC InicioRecPiezas AT %M3.3, 1 s
   "InicioCinta1" : Bool = PLC InicioCinta1 AT %M3.4, 1 s
   "InicioCinta2" : Bool = PLC InicioCinta2 AT %M3.5, 1 s
   "SolMarchaFin" : Bool = PLC SolMarchaFin AT %M3.6, 1 s
   "IniMarchaFin" : Bool = PLC IniMarchaFin AT %M3.7, 1 s
   "FinMarchaFin" : Bool = PLC FinMarchaFin AT %M4.0, 1 s
   "Emergencia" : Bool = PLC Emergencia AT %M4.1, 1 s
   "PararCintaEntrada" : Bool = PLC PararCintaEntrada AT %M4.3, 1 s
   "Timer1" : Bool = PLC Timer1 AT %M4.7, 1 s
   "Cont01" : Bool = PLC Cont01 AT %M5.0, 1 s
   "Cont02" : Bool = PLC Cont02 AT %M5.1, 1 s
   "Timer2" : Bool = PLC Timer2 AT %M5.2, 1 s
   "Timer3" : Bool = PLC Timer3 AT %M5.3, 1 s
   "Timer4" : Bool = PLC Timer4 AT %M5.4, 1 s
   "MotorVolteoCaja01Izq" : Bool = PLC MotorVolteoCaja01Izq AT %Q0.0, 1 s
   "MotorVolteoCaja01Dch" : Bool = PLC MotorVolteoCaja01Dch AT %Q0.1, 1 s
   "MotorVolteoCaja02Izq" : Bool = PLC MotorVolteoCaja02Izq AT %Q0.2, 1 s
   "MotorVolteoCaja02Dch" : Bool = PLC MotorVolteoCaja02Dch AT %Q0.3, 1 s
   "MotorCilindroRec" : Bool = PLC MotorCilindroRec AT %Q0.4, 1 s
   "MotorCilindroExt" : Bool = PLC MotorCilindroExt AT %Q0.5, 1 s
   "MotorCinta01" : Bool = PLC MotorCinta01 AT %Q0.6, 1 s
   "MotorCinta02" : Bool = PLC MotorCinta02 AT %Q0.7, 1 s
   "MotorCintaEntradaAdelante" : Bool = PLC MotorCintaEntradaAdelante AT %Q1.0, 1 s
   "MotorCintaEntradaAtras" : Bool = PLC MotorCintaEntradaAtras AT %Q1.1, 1 s
   "LV" : Bool = PLC LV AT %Q1.2, 1 s
   "LN" : Bool = PLC LN AT %Q1.3, 1 s
   "LR" : Bool = PLC LR AT %Q1.4, 1 s
   "LE" : Bool = PLC LE AT %Q1.5, 1 s
   "Sirena" : Bool = PLC Sirena AT %Q1.6, 1 s
   "ContCaja01_CV" : Int = PLC ContCaja01.CV, 1 s
   "ContCaja02_CV" : Int = PLC ContCaja02.CV, 1 s

text list "Nombre_imagen_lista_texto": 1 'Imagen raíz'

Template "Plantilla_1" 800x480
   Button "Salir" at 722,440 size 55x39; TextOff 'Salir'; PictureOff "ExitRuntime_KTP900_Basic_PN_TR"; PictureOn "ExitRuntime_KTP900_Basic_PN_TR"
      on Release: StopRuntime(0)
   Button "Template_Button" at 622,440 size 55x39; TextOff 'Text'
   Button "Template_Button_1" at 522,440 size 55x39; TextOff 'Text'
   Button "Template_Button_2" at 422,440 size 55x39; TextOff 'Text'
   Button "Template_Button_3" at 322,440 size 55x39; TextOff 'Text'
   Button "Template_Button_4" at 222,440 size 55x39; TextOff 'Text'
   Button "Template_Button_5" at 122,440 size 55x39; TextOff 'Text'
   Button "Imagen inicial" at 22,440 size 55x39; TextOff 'Imagen inicial'; PictureOff "NavigateHome_KTP900_Basic_PN_TR"; PictureOn "NavigateHome_KTP900_Basic_PN_TR"
      on Release: ActivateScreen("Imagen raíz", 0)
   SymbolicIOField "Imagen_campo_ES_simbólico" at 2,7 size 691x26; TextOff '0'; TextOn '1'; TextList "Nombre_imagen_lista_texto"
      ProcessValue <- "Número_imagen_variable"
      on Change: ActivateScreenByNumber("Número_imagen_variable", 0)
   DateTimeField "HmiScreenItemData" at 695,20 size 105x20
   DateTimeField "HmiScreenItemData_1" at 695,0 size 105x20

screen "Imagen raíz" 800x480, template "Plantilla_1"
   on GenerateScreen: SetTag("Número_imagen_variable", 1)
   Button "Botón_1" at 478,302 size 38x28; TextOff 'PP'
      on Press: InvertBit("PP")
      Appearance <- "PP"
   Button "Botón_2" at 478,350 size 38x28; TextOff 'PM'
      on Press: InvertBit("PM")
      Appearance <- "PM"
   Button "Botón_3" at 478,398 size 38x28; TextOff 'PR'
      on Press: InvertBit("PR")
      Appearance <- "PR"
   Button "Botón_4" at 478,446 size 38x28; TextOff 'SE'
      on Press: InvertBit("SE")
      Appearance <- "SE"
   GraphicView "Visor de gráficos_2" at 720,249 size 43x39; Picture "Gráfico_2"
      Appearance <- "Sirena"
   Circle "Círculo_1" at 555,329 size 20x20
      Appearance <- "SolCondIni"
   Circle "Círculo_2" at 555,391 size 20x20
      Appearance <- "ParoFC"
   Circle "Círculo_3" at 555,422 size 20x20
      Appearance <- "SolMarchaFin"
   Circle "Círculo_4" at 555,299 size 20x20
      Appearance <- "Inicio"
   TextField "Campo de texto_1" at 586,299 size 54x20; Text 'Inicio'
   TextField "Campo de texto_2" at 586,329 size 181x20; Text 'CondicionesIniciales'
   TextField "Campo de texto_3" at 586,391 size 65x20; Text 'ParoFC'
   TextField "Campo de texto_4" at 586,422 size 120x20; Text 'SolMarchaFin'
   Circle "Círculo_5" at 555,451 size 20x20
      Appearance <- "Emergencia"
   TextField "Campo de texto_5" at 586,449 size 104x25; Text 'Emergencia'
   GraphicView "Visor de gráficos_5" at 98,206 size 59x71; Picture "Gráfico_8"
      Visibility <- "SenCil01Med"
   GraphicView "Visor de gráficos_1" at 272,207 size 59x71; Picture "Gráfico_11"
      Visibility <- "SenCil01Med"
   IOField "Campo ES_1" at 285,180 size 39x23; FormatPattern s99
      ProcessValue <- "ContCaja02_CV"
   IOField "Campo ES_2" at 109,178 size 38x25; FormatPattern s99
      ProcessValue <- "ContCaja01_CV"
   GraphicView "Visor de gráficos_8" at 173,73 size 75x127; Picture "Gráfico_15"
      Appearance <- "MotorCintaEntradaAdelante"
   GraphicView "Visor de gráficos_9" at 273,302 size 53x103; Picture "Gráfico_15"
      Appearance <- "SenCinta02"
   GraphicView "Visor de gráficos_10" at 104,300 size 52x105; Picture "Gráfico_15"
      Appearance <- "SenCinta01"
   Circle "Círculo_6" at 562,254 size 31x31
      Appearance <- "LN"
   Circle "Círculo_7" at 638,254 size 31x31
      Appearance <- "LE"
   Circle "Círculo_8" at 478,254 size 31x31
      Appearance <- "LV"
   TextField "Campo de texto_6" at 562,254 size 31x31; Text 'LN'
   TextField "Campo de texto_7" at 478,254 size 31x31; Text 'LV'
   TextField "Campo de texto_8" at 638,254 size 31x31; Text 'LE'
   Button "Botón_8" at 164,35 size 94x26; TextOff 'SenCintaEntrada'
      on Press: InvertBit("SenCintaEntrada")
      Appearance <- "SenCintaEntrada"
   Button "Botón_5" at 341,175 size 97x27; TextOff 'Caja02PosIni'
      on Press: InvertBit("SenCaja02PosIni")
      Appearance <- "SenCaja02PosIni"
   Button "Botón_9" at 5,176 size 100x25; TextOff 'Caja01PosIni'
      on Press: InvertBit("SenCaja01PosIni")
      Appearance <- "SenCaja01PosIni"
   TextField "Campo de texto_9" at 106,163 size 42x15; Text 'Caja01'
   TextField "Campo de texto_10" at 281,165 size 42x15; Text 'Caja02'
   Button "Botón_10" at 81,410 size 107x32; TextOff 'SenCinta01'
      on Press: InvertBit("SenCinta01")
      Appearance <- "SenCinta01"
   Button "Botón_11" at 253,410 size 108x32; TextOff 'SenCinta02'
      on Press: InvertBit("SenCinta02")
      Appearance <- "SenCinta02"
   Circle "Círculo_9" at 341,120 size 35x35
      Appearance <- "MotorCilindroRec"
   Circle "Círculo_11" at 398,119 size 35x35
      Appearance <- "MotorCilindroExt"
   TextField "Campo de texto_11" at 346,130 size 25x15; Text 'REC'
   TextField "Campo de texto_13" at 403,129 size 25x15; Text 'EXT'
   Button "Botón_12" at 87,275 size 86x24; TextOff 'Caja01Volteada'
      on Press: InvertBit("SenIndCaja01")
      Appearance <- "SenIndCaja01"
   GraphicView "Visor de gráficos_3" at 186,206 size 59x71; Picture "Gráfico_11"
      Visibility <- "SenCil01Ext"
   GraphicView "Visor de gráficos_4" at 361,207 size 59x71; Picture "Gráfico_11"
      Visibility <- "SenCil01Ext"
   GraphicView "Visor de gráficos_6" at 11,206 size 59x71; Picture "Gráfico_11"
      Visibility <- "SenCil01Rec"
   GraphicView "Visor de gráficos_7" at 187,206 size 59x71; Picture "Gráfico_11"
      Visibility <- "SenCil01Rec"
   TextField "Campo de texto_14" at 315,89 size 149x23; Text 'Estado del Motor:'
   Button "Botón_13" at 256,275 size 88x25; TextOff 'Caja02Volteada'
      on Press: InvertBit("SenIndCaja02")
      Appearance <- "SenIndCaja02"
   Circle "Círculo_12" at 555,360 size 20x20
      Appearance <- "ProdNorm"
   TextField "Campo de texto_15" at 586,360 size 163x20; Text 'ProducciónNormal'
   Button "Botón_15" at 487,123 size 52x27; TextOff 'Rec'
      Appearance <- "SenCil01Rec"
      on Press: InvertBit("SenCil01Rec")
   TextField "Campo de texto_12" at 488,88 size 161x23; Text 'Estado del cilindro:'
   Button "Botón_16" at 547,123 size 52x27; TextOff 'Med'
      on Press: InvertBit("SenCil01Med")
      Appearance <- "SenCil01Med"
   Button "Botón_17" at 608,123 size 52x27; TextOff 'Ext'
      on Press: InvertBit("SenCil01Ext")
      Appearance <- "SenCil01Ext"
   GraphicView "Visor de gráficos_11" at 184,124 size 101x52; Picture "Gráfico_1"
      Appearance <- "FCInferior"
   GraphicView "Visor de gráficos_12" at 180,113 size 121x48; Picture "Gráfico_3"
      Appearance <- "FCSuperior"
   TextField "Campo de texto_21" at 683,250 size 35x32; Text '((('
      Appearance <- "Sirena"
      Visibility <- "Sirena"
   GraphicView "Visor de gráficos_13" at 165,220 size 23x26; Picture "pngwing.com_1"
      Visibility <- "MotorVolteoCaja01Izq"
   GraphicView "Visor de gráficos_14" at 70,222 size 26x24; Picture "pngwing.com"
      Visibility <- "MotorVolteoCaja01Dch"
   GraphicView "Visor de gráficos_15" at 245,227 size 26x24; Picture "pngwing.com"
      Visibility <- "MotorVolteoCaja02Dch"
   GraphicView "Visor de gráficos_16" at 338,228 size 23x26; Picture "pngwing.com_1"
      Visibility <- "MotorVolteoCaja02Izq"
   GraphicView "Visor de gráficos_17" at 147,137 size 36x30; Picture "Gráfico_7"
      Visibility <- "MotorCintaEntradaAdelante"
   GraphicView "Visor de gráficos_18" at 147,93 size 36x30; Picture "Gráfico_9"
      Visibility <- "MotorCintaEntradaAtras"
   Button "Botón_6" at 272,134 size 15x15; TextOff 'Text'
      on Press: InvertBit("FCSuperior"); InvertBit("FCInferior")
      Appearance <- "FCSuperior"
   Button "Botón_7" at 257,154 size 15x15; TextOff 'Text'
      on Press: InvertBit("FCInferior")
      Appearance <- "FCInferior"
*)